// TIA Portal V16 export
// export: Created 2021-11-12T13:31:59.2910616Z, ExportSetting WithDefaults, DisplayName Totally Integrated Automation Portal, DisplayVersion V16 Update 3, DisplayName TIA Portal Version Control Interface, DisplayVersion V16 Update 2, DisplayName TIA Portal Openness, DisplayVersion V16 Update 3, DisplayName SINAMICS Startdrive Advanced, DisplayVersion V16 Update 5, DisplayName SINAMICS Startdrive G130, G150, S120, S150, SINAMICS MV, S210, DisplayVersion V16 Update 5, DisplayName SINAMICS Startdrive G110M, G120, G120C, G120D, G120P, G115D, DisplayVersion V16 Update 5, DisplayName STEP 7 Professional, DisplayVersion V16 Update 3, DisplayName STEP 7 Safety, DisplayVersion V16, DisplayName WinCC UA Professional, DisplayVersion V16 Update 3
FUNCTION_BLOCK "Zone100"   // FB71, LAD
{ S7_Optimized_Access := 'TRUE' }
VERSION : 0.1
// stored: AutoNumber false, IsIECCheckEnabled false, IsRetainMemResEnabled false, MemoryReserve 100, SetENOAutomatically false, UDAEnableTagReadback false
   VAR
      SF_ZoneMode { S7_SetPoint := 'True'} : "STD_Zone";
      SF_StationKAS1Mode { S7_SetPoint := 'True'} : "STD_Station";
      SF_StationKAS2Mode { S7_SetPoint := 'True'} : "STD_Station";
      SF_Station110Mode { S7_SetPoint := 'True'} : "STD_Station";
      SF_Station120Mode { S7_SetPoint := 'True'} : "STD_Station";
      SF_Station1R1Mode { S7_SetPoint := 'True'} : "STD_Station";
      SF_Station1R2Mode { S7_SetPoint := 'True'} : "STD_Station";
      SF_Station130Mode { S7_SetPoint := 'True'} : "STD_Station";
      SF_Station140Mode { S7_SetPoint := 'True'} : "STD_Station";
      SF_Station1R3Mode { S7_SetPoint := 'True'} : "STD_Station";
      SF_Station1R4Mode { S7_SetPoint := 'True'} : "STD_Station";
      SF_Station150Mode { S7_SetPoint := 'True'} : "STD_Station";
      SF_Station160Mode { S7_SetPoint := 'True'} : "STD_Station";
      SF_Station170Mode { S7_SetPoint := 'True'} : "STD_Station";
      SF_Station180Mode { S7_SetPoint := 'True'} : "STD_Station";
      SF_Station1R5Mode { S7_SetPoint := 'True'} : "STD_Station";
      SF_Station1R6Mode { S7_SetPoint := 'True'} : "STD_Station";
      SF_StationBSN1Mode { S7_SetPoint := 'True'} : "STD_Station";
      SF_StationBSN2Mode { S7_SetPoint := 'True'} : "STD_Station";
      SF_CameraLights { S7_SetPoint := 'True'} : "STD_OnOff";
      ST_TONZone1ServModeAct { S7_SetPoint := 'True'} : TON_TIME;   // Timer for Zone 100 service mode
      SS_Edge { S7_SetPoint := 'True'} : Array[0..100] of Bool;
   END_VAR
   VAR_TEMP
      TS_Zone : "UDT_ZoneControl";
      TS_StationKAS1 : "UDT_StationControl";
      TS_StationKAS2 : "UDT_StationControl";
      TS_Station110 : "UDT_StationControl";
      TS_Station120 : "UDT_StationControl";
      TS_Station1R1 : "UDT_StationControl";
      TS_Station1R2 : "UDT_StationControl";
      TS_Station130 : "UDT_StationControl";
      TS_Station140 : "UDT_StationControl";
      TS_Station1R3 : "UDT_StationControl";
      TS_Station1R4 : "UDT_StationControl";
      TS_Station150 : "UDT_StationControl";
      TS_Station160 : "UDT_StationControl";
      TS_Station170 : "UDT_StationControl";
      TS_Station180 : "UDT_StationControl";
      TS_Station1R5 : "UDT_StationControl";
      TS_Station1R6 : "UDT_StationControl";
      TS_StationBSN1 : "UDT_StationControl";
      TS_StationBSN2 : "UDT_StationControl";
      TB1AckFlt1 : Bool;   // LED - acknowledge error button
      TB1AckFlt2 : Bool;   // LED - acknowledge error button
      TB1AckFlt3 : Bool;   // LED - acknowledge error button
      TB1AckSafety1 : Bool;   // LED - acknowledge safety button
      TB1AckSafety2 : Bool;   // LED - acknowledge safety button
      TB1AckSafety3 : Bool;   // LED - acknowledge safety button
      TB1AutStart1 : Bool;   // LED - automat start button
      TB1AutStart2 : Bool;   // LED - automat start button
      TB1AutStart3 : Bool;   // LED - automat start button
      TB1SigRed1 : Bool;   // Light signal - red
      TB1SigRed2 : Bool;   // Light signal - red
      TB1SigRed3 : Bool;   // Light signal - red
      TB1SigYlw1 : Bool;   // Light signal - yellow
      TB1SigYlw2 : Bool;   // Light signal - yellow
      TB1SigYlw3 : Bool;   // Light signal - yellow
      TB1SigGrn1 : Bool;   // Light signal - green
      TB1SigGrn2 : Bool;   // Light signal - green
      TB1SigGrn3 : Bool;   // Light signal - green
      TB1SigAcs1 : Bool;   // Acustic signal
      TB1SigAcs2 : Bool;   // Acustic signal
      TB1SigAcs3 : Bool;   // Acustic signal
      TB1Sig110AutStart : Bool;   // Station 110 run bulb
      TB1Sig110Man : Bool;   // Station 110 manual mode bulb
      TB1Sig110Rem : Bool;   // Station 110 remote mode bulb
      TB1Sig120AutStart : Bool;   // Station 120 run bulb
      TB1Sig120Man : Bool;   // Station 120 manual mode bulb
      TB1Sig120Rem : Bool;   // Station 120 remote mode bulb
      TB1Bin : Bool;   // Something is missing
      TB1CameraLightsON : Bool;
      TB1ReqEndOfCycle : Bool;
      TB1ReqEndOfProd : Bool;
      TB1_1R1AutoOnPE : Bool;   // AutoOn pos edge
      TB1_1R2AutoOnPE : Bool;   // AutoOn pos edge
      TB1_1R3AutoOnPE : Bool;   // AutoOn pos edge
      TB1_1R4AutoOnPE : Bool;   // AutoOn pos edge
      TB1_1R5AutoOnPE : Bool;   // AutoOn pos edge
      TB1_1R6AutoOnPE : Bool;   // AutoOn pos edge
      TB1_1R1AutoOnNE : Bool;   // AutoOn neg edge
      TB1_1R2AutoOnNE : Bool;   // AutoOn neg edge
      TB1_1R3AutoOnNE : Bool;   // AutoOn neg edge
      TB1_1R4AutoOnNE : Bool;   // AutoOn neg edge
      TB1_1R5AutoOnNE : Bool;   // AutoOn neg edge
      TB1_1R6AutoOnNE : Bool;   // AutoOn neg edge
   END_VAR
   VAR_TEMP   // added for the SCL form of the ladder/FBD networks
      _w1 : Bool;
      _w2 : Bool;
      _w3 : Bool;
   END_VAR
BEGIN

REGION Network 1: *************** Zone 100 ***************
END_REGION

REGION Network 2: Zone 100 - Automat switch HMI command from zone to stations
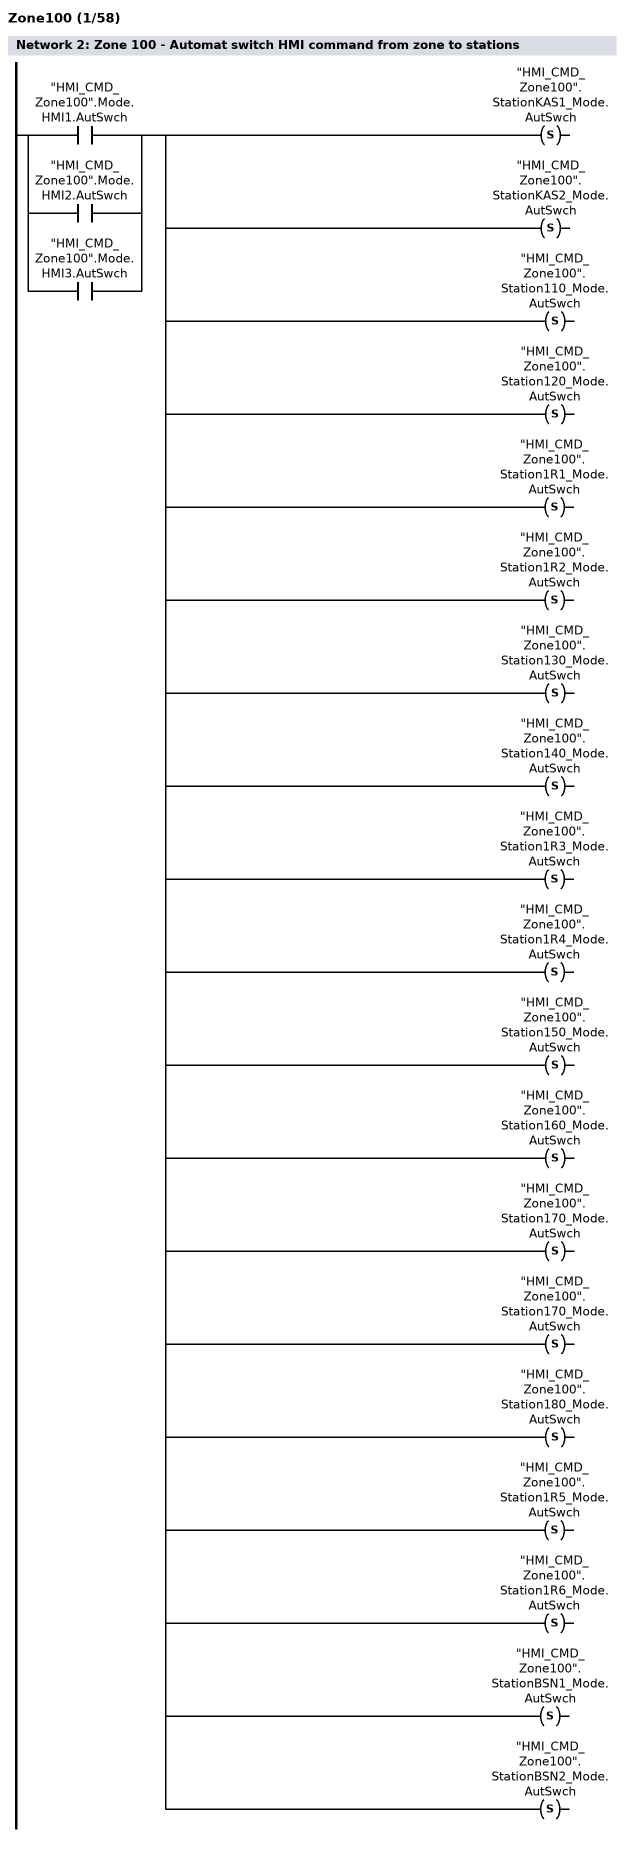
   RUNG wire#powerrail
      Contact( "HMI_CMD_Zone100".Mode.HMI1.AutSwch )
      wire#w1
      S_Coil( "HMI_CMD_Zone100".StationKAS1_Mode.AutSwch )
   END_RUNG
   RUNG wire#powerrail
      Contact( "HMI_CMD_Zone100".Mode.HMI2.AutSwch )
   END_RUNG wire#w1
   RUNG wire#powerrail
      Contact( "HMI_CMD_Zone100".Mode.HMI3.AutSwch )
   END_RUNG wire#w1
   RUNG wire#w1
      S_Coil( "HMI_CMD_Zone100".StationKAS2_Mode.AutSwch )
   END_RUNG
   RUNG wire#w1
      S_Coil( "HMI_CMD_Zone100".Station110_Mode.AutSwch )
   END_RUNG
   RUNG wire#w1
      S_Coil( "HMI_CMD_Zone100".Station120_Mode.AutSwch )
   END_RUNG
   RUNG wire#w1
      S_Coil( "HMI_CMD_Zone100".Station1R1_Mode.AutSwch )
   END_RUNG
   RUNG wire#w1
      S_Coil( "HMI_CMD_Zone100".Station1R2_Mode.AutSwch )
   END_RUNG
   RUNG wire#w1
      S_Coil( "HMI_CMD_Zone100".Station130_Mode.AutSwch )
   END_RUNG
   RUNG wire#w1
      S_Coil( "HMI_CMD_Zone100".Station140_Mode.AutSwch )
   END_RUNG
   RUNG wire#w1
      S_Coil( "HMI_CMD_Zone100".Station1R3_Mode.AutSwch )
   END_RUNG
   RUNG wire#w1
      S_Coil( "HMI_CMD_Zone100".Station1R4_Mode.AutSwch )
   END_RUNG
   RUNG wire#w1
      S_Coil( "HMI_CMD_Zone100".Station150_Mode.AutSwch )
   END_RUNG
   RUNG wire#w1
      S_Coil( "HMI_CMD_Zone100".Station160_Mode.AutSwch )
   END_RUNG
   RUNG wire#w1
      S_Coil( "HMI_CMD_Zone100".Station170_Mode.AutSwch )
   END_RUNG
   RUNG wire#w1
      S_Coil( "HMI_CMD_Zone100".Station170_Mode.AutSwch )
   END_RUNG
   RUNG wire#w1
      S_Coil( "HMI_CMD_Zone100".Station180_Mode.AutSwch )
   END_RUNG
   RUNG wire#w1
      S_Coil( "HMI_CMD_Zone100".Station1R5_Mode.AutSwch )
   END_RUNG
   RUNG wire#w1
      S_Coil( "HMI_CMD_Zone100".Station1R6_Mode.AutSwch )
   END_RUNG
   RUNG wire#w1
      S_Coil( "HMI_CMD_Zone100".StationBSN1_Mode.AutSwch )
   END_RUNG
   RUNG wire#w1
      S_Coil( "HMI_CMD_Zone100".StationBSN2_Mode.AutSwch )
   END_RUNG
   // the same network as SCL:
   IF "HMI_CMD_Zone100".Mode.HMI1.AutSwch OR "HMI_CMD_Zone100".Mode.HMI2.AutSwch OR "HMI_CMD_Zone100".Mode.HMI3.AutSwch THEN
       "HMI_CMD_Zone100".StationKAS1_Mode.AutSwch := TRUE;
       "HMI_CMD_Zone100".StationKAS2_Mode.AutSwch := TRUE;
       "HMI_CMD_Zone100".Station110_Mode.AutSwch := TRUE;
       "HMI_CMD_Zone100".Station120_Mode.AutSwch := TRUE;
       "HMI_CMD_Zone100".Station1R1_Mode.AutSwch := TRUE;
       "HMI_CMD_Zone100".Station1R2_Mode.AutSwch := TRUE;
       "HMI_CMD_Zone100".Station130_Mode.AutSwch := TRUE;
       "HMI_CMD_Zone100".Station140_Mode.AutSwch := TRUE;
       "HMI_CMD_Zone100".Station1R3_Mode.AutSwch := TRUE;
       "HMI_CMD_Zone100".Station1R4_Mode.AutSwch := TRUE;
       "HMI_CMD_Zone100".Station150_Mode.AutSwch := TRUE;
       "HMI_CMD_Zone100".Station160_Mode.AutSwch := TRUE;
       "HMI_CMD_Zone100".Station170_Mode.AutSwch := TRUE;
       "HMI_CMD_Zone100".Station170_Mode.AutSwch := TRUE;
       "HMI_CMD_Zone100".Station180_Mode.AutSwch := TRUE;
       "HMI_CMD_Zone100".Station1R5_Mode.AutSwch := TRUE;
       "HMI_CMD_Zone100".Station1R6_Mode.AutSwch := TRUE;
       "HMI_CMD_Zone100".StationBSN1_Mode.AutSwch := TRUE;
       "HMI_CMD_Zone100".StationBSN2_Mode.AutSwch := TRUE;
   END_IF;
END_REGION

REGION Network 3: Zone 100 - Manual switch HMI command from zone to stations
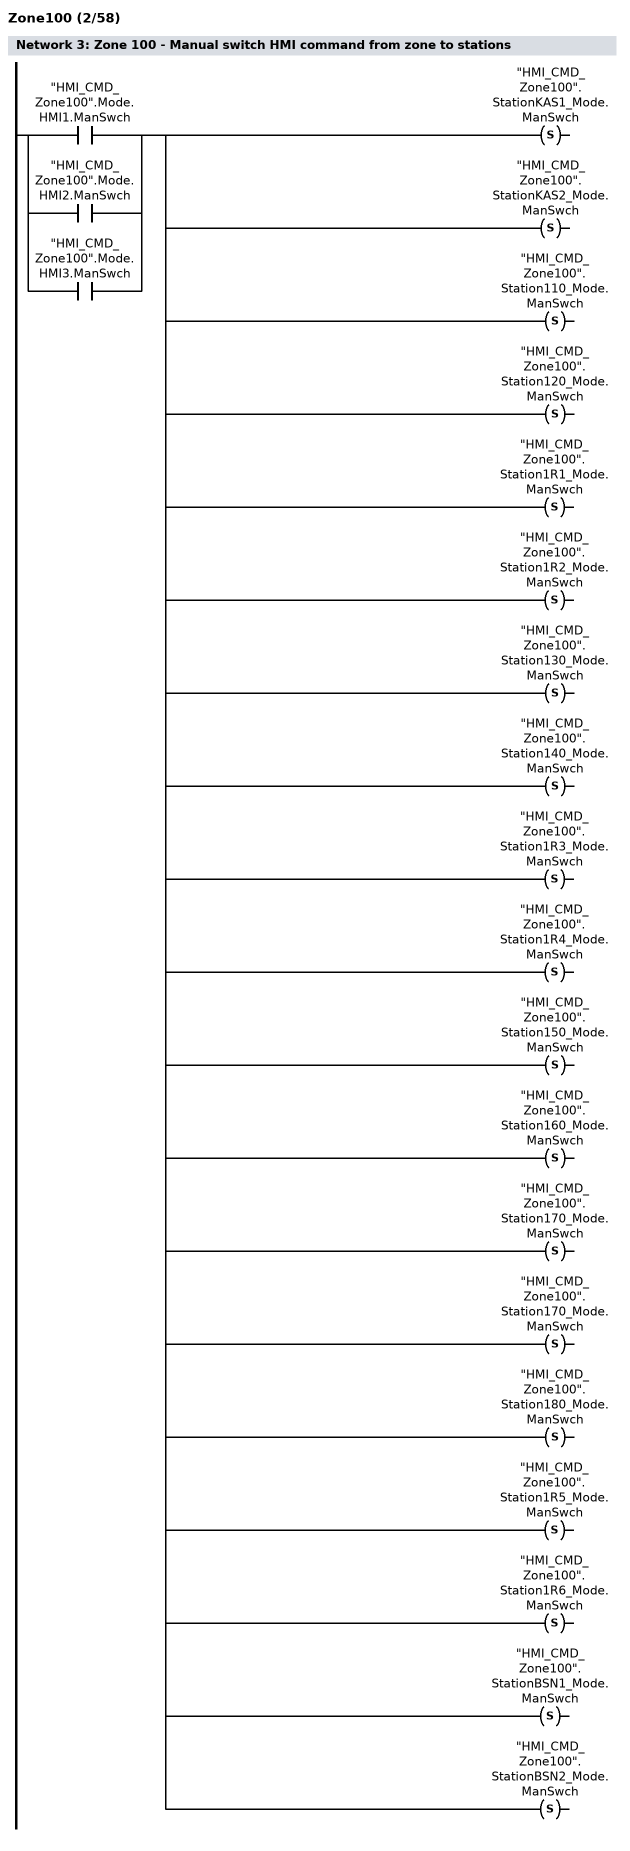
   RUNG wire#powerrail
      Contact( "HMI_CMD_Zone100".Mode.HMI1.ManSwch )
      wire#w1
      S_Coil( "HMI_CMD_Zone100".StationKAS1_Mode.ManSwch )
   END_RUNG
   RUNG wire#powerrail
      Contact( "HMI_CMD_Zone100".Mode.HMI2.ManSwch )
   END_RUNG wire#w1
   RUNG wire#powerrail
      Contact( "HMI_CMD_Zone100".Mode.HMI3.ManSwch )
   END_RUNG wire#w1
   RUNG wire#w1
      S_Coil( "HMI_CMD_Zone100".StationKAS2_Mode.ManSwch )
   END_RUNG
   RUNG wire#w1
      S_Coil( "HMI_CMD_Zone100".Station110_Mode.ManSwch )
   END_RUNG
   RUNG wire#w1
      S_Coil( "HMI_CMD_Zone100".Station120_Mode.ManSwch )
   END_RUNG
   RUNG wire#w1
      S_Coil( "HMI_CMD_Zone100".Station1R1_Mode.ManSwch )
   END_RUNG
   RUNG wire#w1
      S_Coil( "HMI_CMD_Zone100".Station1R2_Mode.ManSwch )
   END_RUNG
   RUNG wire#w1
      S_Coil( "HMI_CMD_Zone100".Station130_Mode.ManSwch )
   END_RUNG
   RUNG wire#w1
      S_Coil( "HMI_CMD_Zone100".Station140_Mode.ManSwch )
   END_RUNG
   RUNG wire#w1
      S_Coil( "HMI_CMD_Zone100".Station1R3_Mode.ManSwch )
   END_RUNG
   RUNG wire#w1
      S_Coil( "HMI_CMD_Zone100".Station1R4_Mode.ManSwch )
   END_RUNG
   RUNG wire#w1
      S_Coil( "HMI_CMD_Zone100".Station150_Mode.ManSwch )
   END_RUNG
   RUNG wire#w1
      S_Coil( "HMI_CMD_Zone100".Station160_Mode.ManSwch )
   END_RUNG
   RUNG wire#w1
      S_Coil( "HMI_CMD_Zone100".Station170_Mode.ManSwch )
   END_RUNG
   RUNG wire#w1
      S_Coil( "HMI_CMD_Zone100".Station170_Mode.ManSwch )
   END_RUNG
   RUNG wire#w1
      S_Coil( "HMI_CMD_Zone100".Station180_Mode.ManSwch )
   END_RUNG
   RUNG wire#w1
      S_Coil( "HMI_CMD_Zone100".Station1R5_Mode.ManSwch )
   END_RUNG
   RUNG wire#w1
      S_Coil( "HMI_CMD_Zone100".Station1R6_Mode.ManSwch )
   END_RUNG
   RUNG wire#w1
      S_Coil( "HMI_CMD_Zone100".StationBSN1_Mode.ManSwch )
   END_RUNG
   RUNG wire#w1
      S_Coil( "HMI_CMD_Zone100".StationBSN2_Mode.ManSwch )
   END_RUNG
   // the same network as SCL:
   IF "HMI_CMD_Zone100".Mode.HMI1.ManSwch OR "HMI_CMD_Zone100".Mode.HMI2.ManSwch OR "HMI_CMD_Zone100".Mode.HMI3.ManSwch THEN
       "HMI_CMD_Zone100".StationKAS1_Mode.ManSwch := TRUE;
       "HMI_CMD_Zone100".StationKAS2_Mode.ManSwch := TRUE;
       "HMI_CMD_Zone100".Station110_Mode.ManSwch := TRUE;
       "HMI_CMD_Zone100".Station120_Mode.ManSwch := TRUE;
       "HMI_CMD_Zone100".Station1R1_Mode.ManSwch := TRUE;
       "HMI_CMD_Zone100".Station1R2_Mode.ManSwch := TRUE;
       "HMI_CMD_Zone100".Station130_Mode.ManSwch := TRUE;
       "HMI_CMD_Zone100".Station140_Mode.ManSwch := TRUE;
       "HMI_CMD_Zone100".Station1R3_Mode.ManSwch := TRUE;
       "HMI_CMD_Zone100".Station1R4_Mode.ManSwch := TRUE;
       "HMI_CMD_Zone100".Station150_Mode.ManSwch := TRUE;
       "HMI_CMD_Zone100".Station160_Mode.ManSwch := TRUE;
       "HMI_CMD_Zone100".Station170_Mode.ManSwch := TRUE;
       "HMI_CMD_Zone100".Station170_Mode.ManSwch := TRUE;
       "HMI_CMD_Zone100".Station180_Mode.ManSwch := TRUE;
       "HMI_CMD_Zone100".Station1R5_Mode.ManSwch := TRUE;
       "HMI_CMD_Zone100".Station1R6_Mode.ManSwch := TRUE;
       "HMI_CMD_Zone100".StationBSN1_Mode.ManSwch := TRUE;
       "HMI_CMD_Zone100".StationBSN2_Mode.ManSwch := TRUE;
   END_IF;
END_REGION

REGION Network 4: Zone 100 - Off switch HMI command from zone to stations
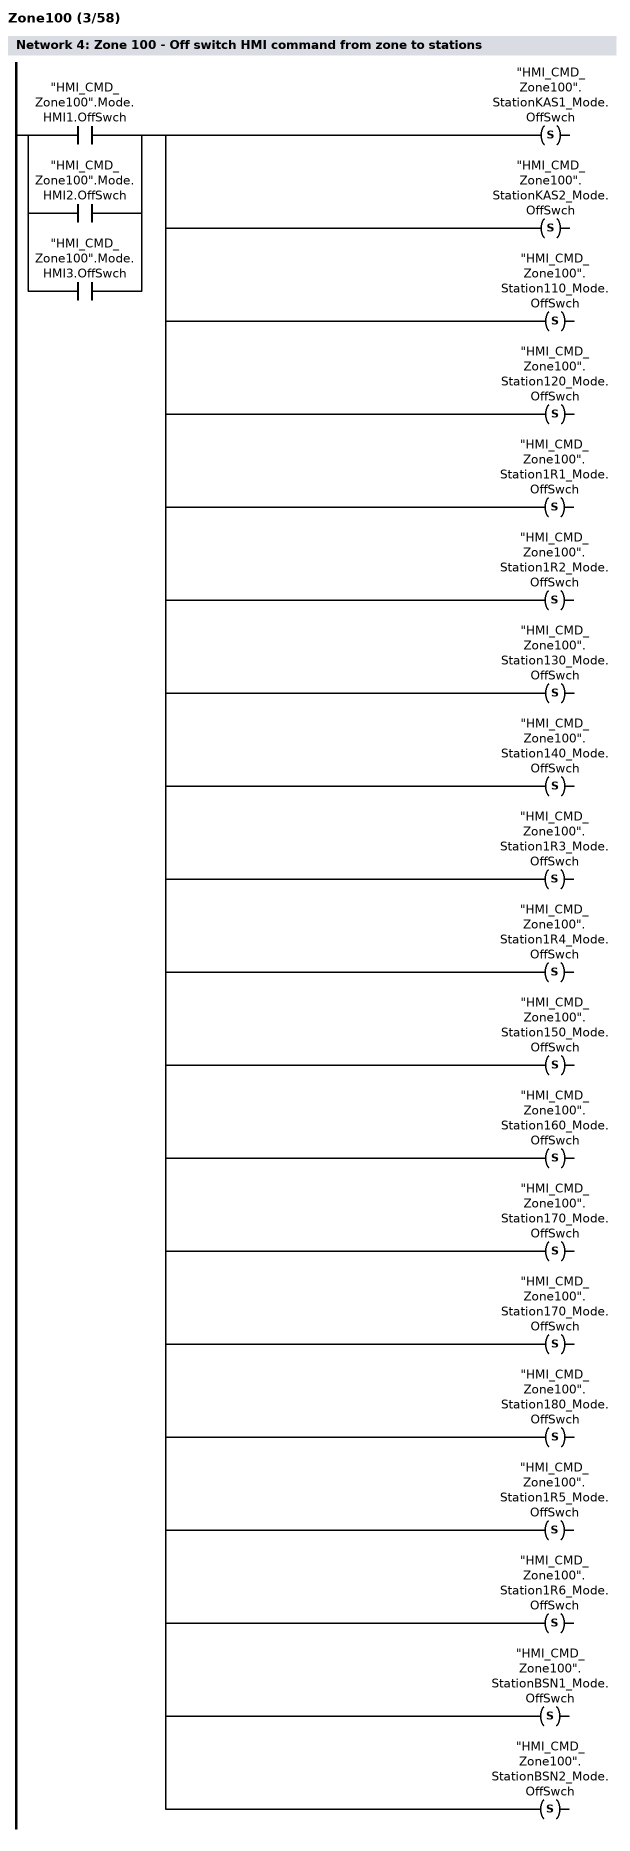
   RUNG wire#powerrail
      Contact( "HMI_CMD_Zone100".Mode.HMI1.OffSwch )
      wire#w1
      S_Coil( "HMI_CMD_Zone100".StationKAS1_Mode.OffSwch )
   END_RUNG
   RUNG wire#powerrail
      Contact( "HMI_CMD_Zone100".Mode.HMI2.OffSwch )
   END_RUNG wire#w1
   RUNG wire#powerrail
      Contact( "HMI_CMD_Zone100".Mode.HMI3.OffSwch )
   END_RUNG wire#w1
   RUNG wire#w1
      S_Coil( "HMI_CMD_Zone100".StationKAS2_Mode.OffSwch )
   END_RUNG
   RUNG wire#w1
      S_Coil( "HMI_CMD_Zone100".Station110_Mode.OffSwch )
   END_RUNG
   RUNG wire#w1
      S_Coil( "HMI_CMD_Zone100".Station120_Mode.OffSwch )
   END_RUNG
   RUNG wire#w1
      S_Coil( "HMI_CMD_Zone100".Station1R1_Mode.OffSwch )
   END_RUNG
   RUNG wire#w1
      S_Coil( "HMI_CMD_Zone100".Station1R2_Mode.OffSwch )
   END_RUNG
   RUNG wire#w1
      S_Coil( "HMI_CMD_Zone100".Station130_Mode.OffSwch )
   END_RUNG
   RUNG wire#w1
      S_Coil( "HMI_CMD_Zone100".Station140_Mode.OffSwch )
   END_RUNG
   RUNG wire#w1
      S_Coil( "HMI_CMD_Zone100".Station1R3_Mode.OffSwch )
   END_RUNG
   RUNG wire#w1
      S_Coil( "HMI_CMD_Zone100".Station1R4_Mode.OffSwch )
   END_RUNG
   RUNG wire#w1
      S_Coil( "HMI_CMD_Zone100".Station150_Mode.OffSwch )
   END_RUNG
   RUNG wire#w1
      S_Coil( "HMI_CMD_Zone100".Station160_Mode.OffSwch )
   END_RUNG
   RUNG wire#w1
      S_Coil( "HMI_CMD_Zone100".Station170_Mode.OffSwch )
   END_RUNG
   RUNG wire#w1
      S_Coil( "HMI_CMD_Zone100".Station170_Mode.OffSwch )
   END_RUNG
   RUNG wire#w1
      S_Coil( "HMI_CMD_Zone100".Station180_Mode.OffSwch )
   END_RUNG
   RUNG wire#w1
      S_Coil( "HMI_CMD_Zone100".Station1R5_Mode.OffSwch )
   END_RUNG
   RUNG wire#w1
      S_Coil( "HMI_CMD_Zone100".Station1R6_Mode.OffSwch )
   END_RUNG
   RUNG wire#w1
      S_Coil( "HMI_CMD_Zone100".StationBSN1_Mode.OffSwch )
   END_RUNG
   RUNG wire#w1
      S_Coil( "HMI_CMD_Zone100".StationBSN2_Mode.OffSwch )
   END_RUNG
   // the same network as SCL:
   IF "HMI_CMD_Zone100".Mode.HMI1.OffSwch OR "HMI_CMD_Zone100".Mode.HMI2.OffSwch OR "HMI_CMD_Zone100".Mode.HMI3.OffSwch THEN
       "HMI_CMD_Zone100".StationKAS1_Mode.OffSwch := TRUE;
       "HMI_CMD_Zone100".StationKAS2_Mode.OffSwch := TRUE;
       "HMI_CMD_Zone100".Station110_Mode.OffSwch := TRUE;
       "HMI_CMD_Zone100".Station120_Mode.OffSwch := TRUE;
       "HMI_CMD_Zone100".Station1R1_Mode.OffSwch := TRUE;
       "HMI_CMD_Zone100".Station1R2_Mode.OffSwch := TRUE;
       "HMI_CMD_Zone100".Station130_Mode.OffSwch := TRUE;
       "HMI_CMD_Zone100".Station140_Mode.OffSwch := TRUE;
       "HMI_CMD_Zone100".Station1R3_Mode.OffSwch := TRUE;
       "HMI_CMD_Zone100".Station1R4_Mode.OffSwch := TRUE;
       "HMI_CMD_Zone100".Station150_Mode.OffSwch := TRUE;
       "HMI_CMD_Zone100".Station160_Mode.OffSwch := TRUE;
       "HMI_CMD_Zone100".Station170_Mode.OffSwch := TRUE;
       "HMI_CMD_Zone100".Station170_Mode.OffSwch := TRUE;
       "HMI_CMD_Zone100".Station180_Mode.OffSwch := TRUE;
       "HMI_CMD_Zone100".Station1R5_Mode.OffSwch := TRUE;
       "HMI_CMD_Zone100".Station1R6_Mode.OffSwch := TRUE;
       "HMI_CMD_Zone100".StationBSN1_Mode.OffSwch := TRUE;
       "HMI_CMD_Zone100".StationBSN2_Mode.OffSwch := TRUE;
   END_IF;
END_REGION

REGION Network 5: Zone 100 - change robot tools command
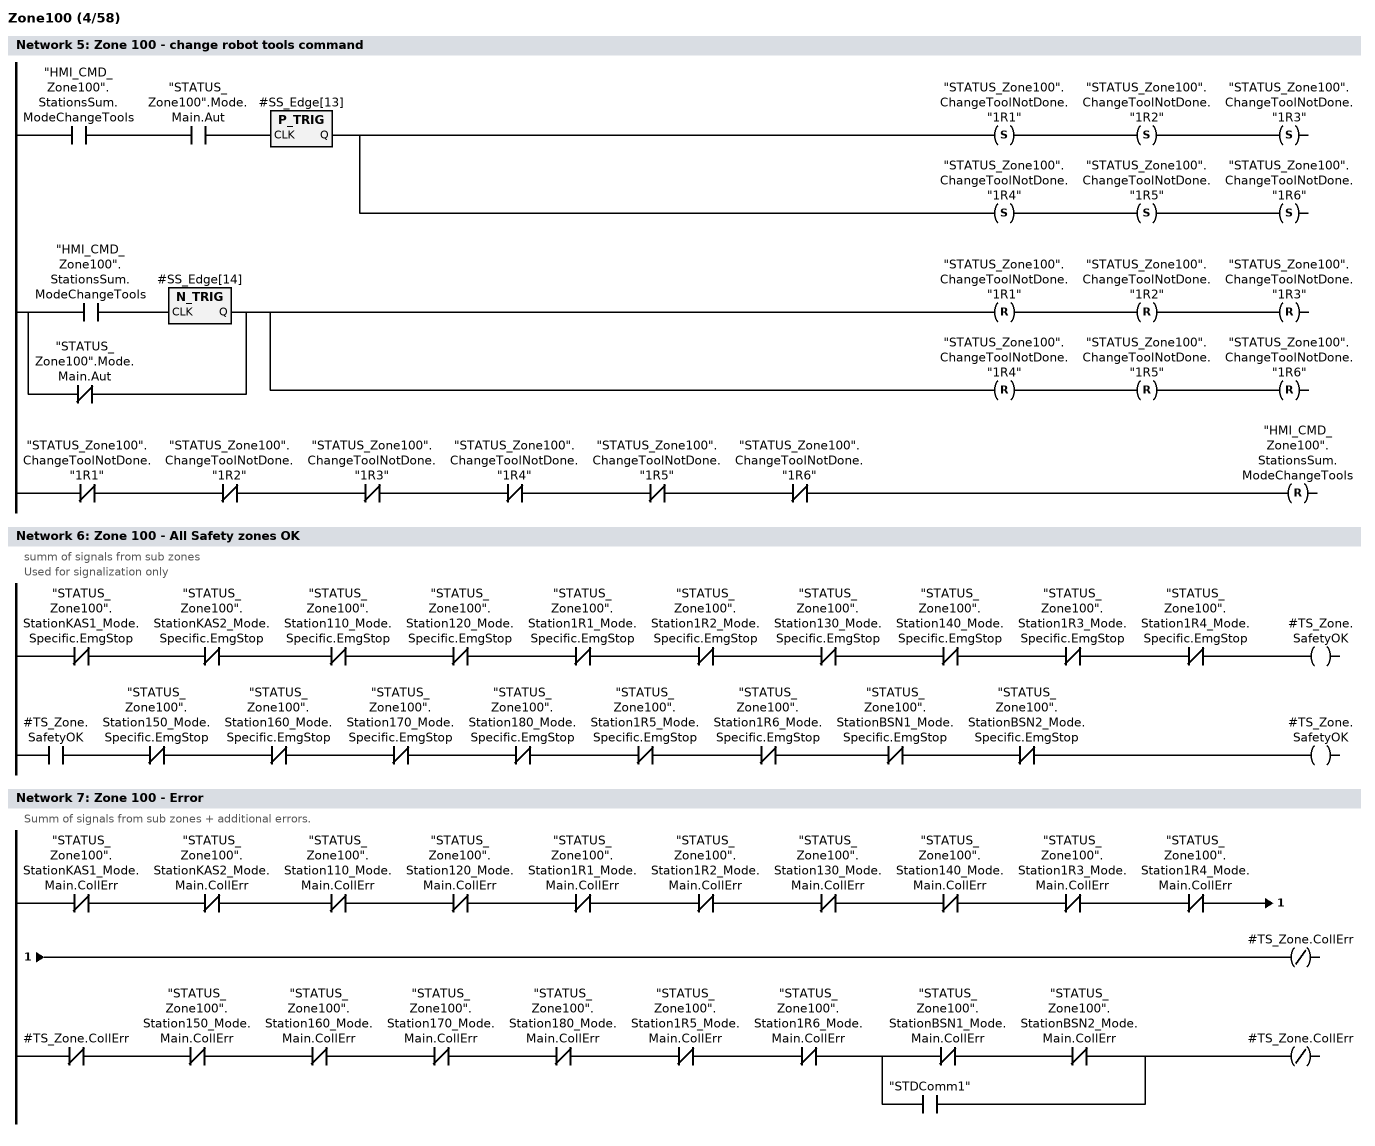
   RUNG wire#powerrail
      Contact( "HMI_CMD_Zone100".StationsSum.ModeChangeTools )
      Contact( "STATUS_Zone100".Mode.Main.Aut )
      P_Trig( #SS_Edge[13] )
      wire#w1
      S_Coil( "STATUS_Zone100".ChangeToolNotDone."1R1" )
      S_Coil( "STATUS_Zone100".ChangeToolNotDone."1R2" )
      S_Coil( "STATUS_Zone100".ChangeToolNotDone."1R3" )
   END_RUNG
   RUNG wire#w1
      S_Coil( "STATUS_Zone100".ChangeToolNotDone."1R4" )
      S_Coil( "STATUS_Zone100".ChangeToolNotDone."1R5" )
      S_Coil( "STATUS_Zone100".ChangeToolNotDone."1R6" )
   END_RUNG
   RUNG wire#powerrail
      Contact( "HMI_CMD_Zone100".StationsSum.ModeChangeTools )
      N_Trig( #SS_Edge[14] )
      wire#w2
      R_Coil( "STATUS_Zone100".ChangeToolNotDone."1R1" )
      R_Coil( "STATUS_Zone100".ChangeToolNotDone."1R2" )
      R_Coil( "STATUS_Zone100".ChangeToolNotDone."1R3" )
   END_RUNG
   RUNG wire#powerrail
      I_Contact( "STATUS_Zone100".Mode.Main.Aut )
   END_RUNG wire#w2
   RUNG wire#w2
      R_Coil( "STATUS_Zone100".ChangeToolNotDone."1R4" )
      R_Coil( "STATUS_Zone100".ChangeToolNotDone."1R5" )
      R_Coil( "STATUS_Zone100".ChangeToolNotDone."1R6" )
   END_RUNG
   RUNG wire#powerrail
      I_Contact( "STATUS_Zone100".ChangeToolNotDone."1R1" )
      I_Contact( "STATUS_Zone100".ChangeToolNotDone."1R2" )
      I_Contact( "STATUS_Zone100".ChangeToolNotDone."1R3" )
      I_Contact( "STATUS_Zone100".ChangeToolNotDone."1R4" )
      I_Contact( "STATUS_Zone100".ChangeToolNotDone."1R5" )
      I_Contact( "STATUS_Zone100".ChangeToolNotDone."1R6" )
      R_Coil( "HMI_CMD_Zone100".StationsSum.ModeChangeTools )
   END_RUNG
   // the same network as SCL:
   #_w1 := "HMI_CMD_Zone100".StationsSum.ModeChangeTools AND "STATUS_Zone100".Mode.Main.Aut;
   #_w2 := #_w1 AND NOT #SS_Edge[13];   // rising edge
   #SS_Edge[13] := #_w1;
   IF #_w2 THEN
       "STATUS_Zone100".ChangeToolNotDone."1R1" := TRUE;
       "STATUS_Zone100".ChangeToolNotDone."1R2" := TRUE;
       "STATUS_Zone100".ChangeToolNotDone."1R3" := TRUE;
       "STATUS_Zone100".ChangeToolNotDone."1R4" := TRUE;
       "STATUS_Zone100".ChangeToolNotDone."1R5" := TRUE;
       "STATUS_Zone100".ChangeToolNotDone."1R6" := TRUE;
   END_IF;
   #_w3 := NOT "HMI_CMD_Zone100".StationsSum.ModeChangeTools AND #SS_Edge[14];   // falling edge
   #SS_Edge[14] := "HMI_CMD_Zone100".StationsSum.ModeChangeTools;
   IF #_w3 OR NOT "STATUS_Zone100".Mode.Main.Aut THEN
       "STATUS_Zone100".ChangeToolNotDone."1R1" := FALSE;
       "STATUS_Zone100".ChangeToolNotDone."1R2" := FALSE;
       "STATUS_Zone100".ChangeToolNotDone."1R3" := FALSE;
       "STATUS_Zone100".ChangeToolNotDone."1R4" := FALSE;
       "STATUS_Zone100".ChangeToolNotDone."1R5" := FALSE;
       "STATUS_Zone100".ChangeToolNotDone."1R6" := FALSE;
   END_IF;
   IF NOT "STATUS_Zone100".ChangeToolNotDone."1R1" AND NOT "STATUS_Zone100".ChangeToolNotDone."1R2" AND NOT "STATUS_Zone100".ChangeToolNotDone."1R3" AND NOT "STATUS_Zone100".ChangeToolNotDone."1R4" AND NOT "STATUS_Zone100".ChangeToolNotDone."1R5" AND NOT "STATUS_Zone100".ChangeToolNotDone."1R6" THEN
       "HMI_CMD_Zone100".StationsSum.ModeChangeTools := FALSE;
   END_IF;
END_REGION

REGION Network 6: Zone 100 - All Safety zones OK
   // summ of signals from sub zones
   // Used for signalization only
   RUNG wire#powerrail
      I_Contact( "STATUS_Zone100".StationKAS1_Mode.Specific.EmgStop )
      I_Contact( "STATUS_Zone100".StationKAS2_Mode.Specific.EmgStop )
      I_Contact( "STATUS_Zone100".Station110_Mode.Specific.EmgStop )
      I_Contact( "STATUS_Zone100".Station120_Mode.Specific.EmgStop )
      I_Contact( "STATUS_Zone100".Station1R1_Mode.Specific.EmgStop )
      I_Contact( "STATUS_Zone100".Station1R2_Mode.Specific.EmgStop )
      I_Contact( "STATUS_Zone100".Station130_Mode.Specific.EmgStop )
      I_Contact( "STATUS_Zone100".Station140_Mode.Specific.EmgStop )
      I_Contact( "STATUS_Zone100".Station1R3_Mode.Specific.EmgStop )
      I_Contact( "STATUS_Zone100".Station1R4_Mode.Specific.EmgStop )
      Coil( #TS_Zone.SafetyOK )
   END_RUNG
   RUNG wire#powerrail
      Contact( #TS_Zone.SafetyOK )
      I_Contact( "STATUS_Zone100".Station150_Mode.Specific.EmgStop )
      I_Contact( "STATUS_Zone100".Station160_Mode.Specific.EmgStop )
      I_Contact( "STATUS_Zone100".Station170_Mode.Specific.EmgStop )
      I_Contact( "STATUS_Zone100".Station180_Mode.Specific.EmgStop )
      I_Contact( "STATUS_Zone100".Station1R5_Mode.Specific.EmgStop )
      I_Contact( "STATUS_Zone100".Station1R6_Mode.Specific.EmgStop )
      I_Contact( "STATUS_Zone100".StationBSN1_Mode.Specific.EmgStop )
      I_Contact( "STATUS_Zone100".StationBSN2_Mode.Specific.EmgStop )
      Coil( #TS_Zone.SafetyOK )
   END_RUNG
   // the same network as SCL:
   #TS_Zone.SafetyOK := NOT "STATUS_Zone100".StationKAS1_Mode.Specific.EmgStop AND NOT "STATUS_Zone100".StationKAS2_Mode.Specific.EmgStop AND NOT "STATUS_Zone100".Station110_Mode.Specific.EmgStop AND NOT "STATUS_Zone100".Station120_Mode.Specific.EmgStop AND NOT "STATUS_Zone100".Station1R1_Mode.Specific.EmgStop AND NOT "STATUS_Zone100".Station1R2_Mode.Specific.EmgStop AND NOT "STATUS_Zone100".Station130_Mode.Specific.EmgStop AND NOT "STATUS_Zone100".Station140_Mode.Specific.EmgStop AND NOT "STATUS_Zone100".Station1R3_Mode.Specific.EmgStop AND NOT "STATUS_Zone100".Station1R4_Mode.Specific.EmgStop;
   #TS_Zone.SafetyOK := #TS_Zone.SafetyOK AND NOT "STATUS_Zone100".Station150_Mode.Specific.EmgStop AND NOT "STATUS_Zone100".Station160_Mode.Specific.EmgStop AND NOT "STATUS_Zone100".Station170_Mode.Specific.EmgStop AND NOT "STATUS_Zone100".Station180_Mode.Specific.EmgStop AND NOT "STATUS_Zone100".Station1R5_Mode.Specific.EmgStop AND NOT "STATUS_Zone100".Station1R6_Mode.Specific.EmgStop AND NOT "STATUS_Zone100".StationBSN1_Mode.Specific.EmgStop AND NOT "STATUS_Zone100".StationBSN2_Mode.Specific.EmgStop;
END_REGION

REGION Network 7: Zone 100 - Error
   // Summ of signals from sub zones + additional errors.
   RUNG wire#powerrail
      I_Contact( "STATUS_Zone100".StationKAS1_Mode.Main.CollErr )
      I_Contact( "STATUS_Zone100".StationKAS2_Mode.Main.CollErr )
      I_Contact( "STATUS_Zone100".Station110_Mode.Main.CollErr )
      I_Contact( "STATUS_Zone100".Station120_Mode.Main.CollErr )
      I_Contact( "STATUS_Zone100".Station1R1_Mode.Main.CollErr )
      I_Contact( "STATUS_Zone100".Station1R2_Mode.Main.CollErr )
      I_Contact( "STATUS_Zone100".Station130_Mode.Main.CollErr )
      I_Contact( "STATUS_Zone100".Station140_Mode.Main.CollErr )
      I_Contact( "STATUS_Zone100".Station1R3_Mode.Main.CollErr )
      I_Contact( "STATUS_Zone100".Station1R4_Mode.Main.CollErr )
      I_Coil( #TS_Zone.CollErr )
   END_RUNG
   RUNG wire#powerrail
      I_Contact( #TS_Zone.CollErr )
      I_Contact( "STATUS_Zone100".Station150_Mode.Main.CollErr )
      I_Contact( "STATUS_Zone100".Station160_Mode.Main.CollErr )
      I_Contact( "STATUS_Zone100".Station170_Mode.Main.CollErr )
      I_Contact( "STATUS_Zone100".Station180_Mode.Main.CollErr )
      I_Contact( "STATUS_Zone100".Station1R5_Mode.Main.CollErr )
      I_Contact( "STATUS_Zone100".Station1R6_Mode.Main.CollErr )
      wire#w1
      I_Contact( "STATUS_Zone100".StationBSN1_Mode.Main.CollErr )
      I_Contact( "STATUS_Zone100".StationBSN2_Mode.Main.CollErr )
      wire#w2
      I_Coil( #TS_Zone.CollErr )
   END_RUNG
   RUNG wire#w1
      Contact( "STDComm1" )
   END_RUNG wire#w2
   // the same network as SCL:
   #TS_Zone.CollErr := NOT (NOT "STATUS_Zone100".StationKAS1_Mode.Main.CollErr AND NOT "STATUS_Zone100".StationKAS2_Mode.Main.CollErr AND NOT "STATUS_Zone100".Station110_Mode.Main.CollErr AND NOT "STATUS_Zone100".Station120_Mode.Main.CollErr AND NOT "STATUS_Zone100".Station1R1_Mode.Main.CollErr AND NOT "STATUS_Zone100".Station1R2_Mode.Main.CollErr AND NOT "STATUS_Zone100".Station130_Mode.Main.CollErr AND NOT "STATUS_Zone100".Station140_Mode.Main.CollErr AND NOT "STATUS_Zone100".Station1R3_Mode.Main.CollErr AND NOT "STATUS_Zone100".Station1R4_Mode.Main.CollErr);
   #TS_Zone.CollErr := NOT (NOT #TS_Zone.CollErr AND NOT "STATUS_Zone100".Station150_Mode.Main.CollErr AND NOT "STATUS_Zone100".Station160_Mode.Main.CollErr AND NOT "STATUS_Zone100".Station170_Mode.Main.CollErr AND NOT "STATUS_Zone100".Station180_Mode.Main.CollErr AND NOT "STATUS_Zone100".Station1R5_Mode.Main.CollErr AND NOT "STATUS_Zone100".Station1R6_Mode.Main.CollErr AND ((NOT "STATUS_Zone100".StationBSN1_Mode.Main.CollErr AND NOT "STATUS_Zone100".StationBSN2_Mode.Main.CollErr) OR "STDComm1"));
END_REGION

REGION Network 8: Zone 100 - Warning
   // Summ of signals from sub zones + additional warnings.
   // Used for signalization only
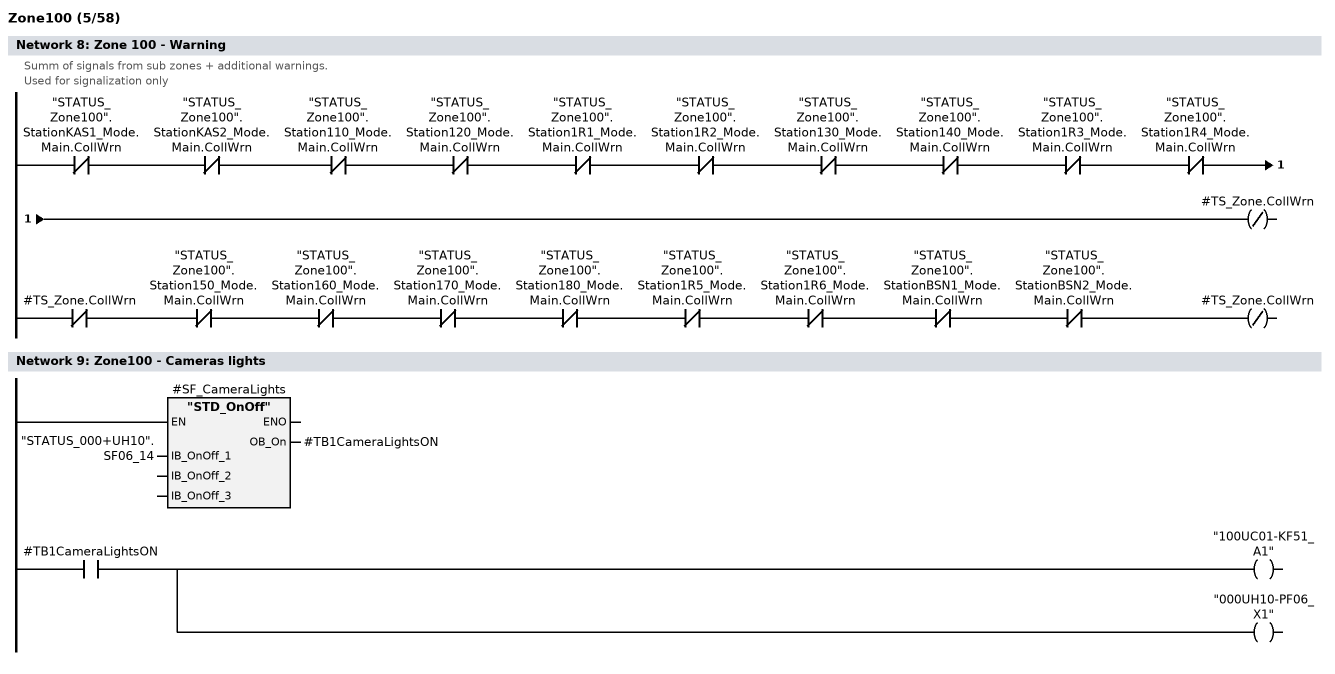
   RUNG wire#powerrail
      I_Contact( "STATUS_Zone100".StationKAS1_Mode.Main.CollWrn )
      I_Contact( "STATUS_Zone100".StationKAS2_Mode.Main.CollWrn )
      I_Contact( "STATUS_Zone100".Station110_Mode.Main.CollWrn )
      I_Contact( "STATUS_Zone100".Station120_Mode.Main.CollWrn )
      I_Contact( "STATUS_Zone100".Station1R1_Mode.Main.CollWrn )
      I_Contact( "STATUS_Zone100".Station1R2_Mode.Main.CollWrn )
      I_Contact( "STATUS_Zone100".Station130_Mode.Main.CollWrn )
      I_Contact( "STATUS_Zone100".Station140_Mode.Main.CollWrn )
      I_Contact( "STATUS_Zone100".Station1R3_Mode.Main.CollWrn )
      I_Contact( "STATUS_Zone100".Station1R4_Mode.Main.CollWrn )
      I_Coil( #TS_Zone.CollWrn )
   END_RUNG
   RUNG wire#powerrail
      I_Contact( #TS_Zone.CollWrn )
      I_Contact( "STATUS_Zone100".Station150_Mode.Main.CollWrn )
      I_Contact( "STATUS_Zone100".Station160_Mode.Main.CollWrn )
      I_Contact( "STATUS_Zone100".Station170_Mode.Main.CollWrn )
      I_Contact( "STATUS_Zone100".Station180_Mode.Main.CollWrn )
      I_Contact( "STATUS_Zone100".Station1R5_Mode.Main.CollWrn )
      I_Contact( "STATUS_Zone100".Station1R6_Mode.Main.CollWrn )
      I_Contact( "STATUS_Zone100".StationBSN1_Mode.Main.CollWrn )
      I_Contact( "STATUS_Zone100".StationBSN2_Mode.Main.CollWrn )
      I_Coil( #TS_Zone.CollWrn )
   END_RUNG
   // the same network as SCL:
   #TS_Zone.CollWrn := NOT (NOT "STATUS_Zone100".StationKAS1_Mode.Main.CollWrn AND NOT "STATUS_Zone100".StationKAS2_Mode.Main.CollWrn AND NOT "STATUS_Zone100".Station110_Mode.Main.CollWrn AND NOT "STATUS_Zone100".Station120_Mode.Main.CollWrn AND NOT "STATUS_Zone100".Station1R1_Mode.Main.CollWrn AND NOT "STATUS_Zone100".Station1R2_Mode.Main.CollWrn AND NOT "STATUS_Zone100".Station130_Mode.Main.CollWrn AND NOT "STATUS_Zone100".Station140_Mode.Main.CollWrn AND NOT "STATUS_Zone100".Station1R3_Mode.Main.CollWrn AND NOT "STATUS_Zone100".Station1R4_Mode.Main.CollWrn);
   #TS_Zone.CollWrn := NOT (NOT #TS_Zone.CollWrn AND NOT "STATUS_Zone100".Station150_Mode.Main.CollWrn AND NOT "STATUS_Zone100".Station160_Mode.Main.CollWrn AND NOT "STATUS_Zone100".Station170_Mode.Main.CollWrn AND NOT "STATUS_Zone100".Station180_Mode.Main.CollWrn AND NOT "STATUS_Zone100".Station1R5_Mode.Main.CollWrn AND NOT "STATUS_Zone100".Station1R6_Mode.Main.CollWrn AND NOT "STATUS_Zone100".StationBSN1_Mode.Main.CollWrn AND NOT "STATUS_Zone100".StationBSN2_Mode.Main.CollWrn);
END_REGION

REGION Network 9: Zone100 - Cameras lights
   RUNG wire#powerrail
      #SF_CameraLights(IB_OnOff_1 := "STATUS_000+UH10".SF06_14, IB_OnOff_2 :=, IB_OnOff_3 :=, OB_On => #TB1CameraLightsON)
   END_RUNG
   RUNG wire#powerrail
      Contact( #TB1CameraLightsON )
      wire#w1
      Coil( "100UC01-KF51_A1" )
   END_RUNG
   RUNG wire#w1
      Coil( "000UH10-PF06_X1" )
   END_RUNG
   // the same network as SCL:
   #SF_CameraLights(IB_OnOff_1 := "STATUS_000+UH10".SF06_14, OB_On => #TB1CameraLightsON);   // "STD_OnOff"
   "100UC01-KF51_A1" := #TB1CameraLightsON;
   "000UH10-PF06_X1" := #TB1CameraLightsON;
END_REGION

REGION Network 10: Zone 100 - All drives running in Automatic
   // Summ of signals from sub zones
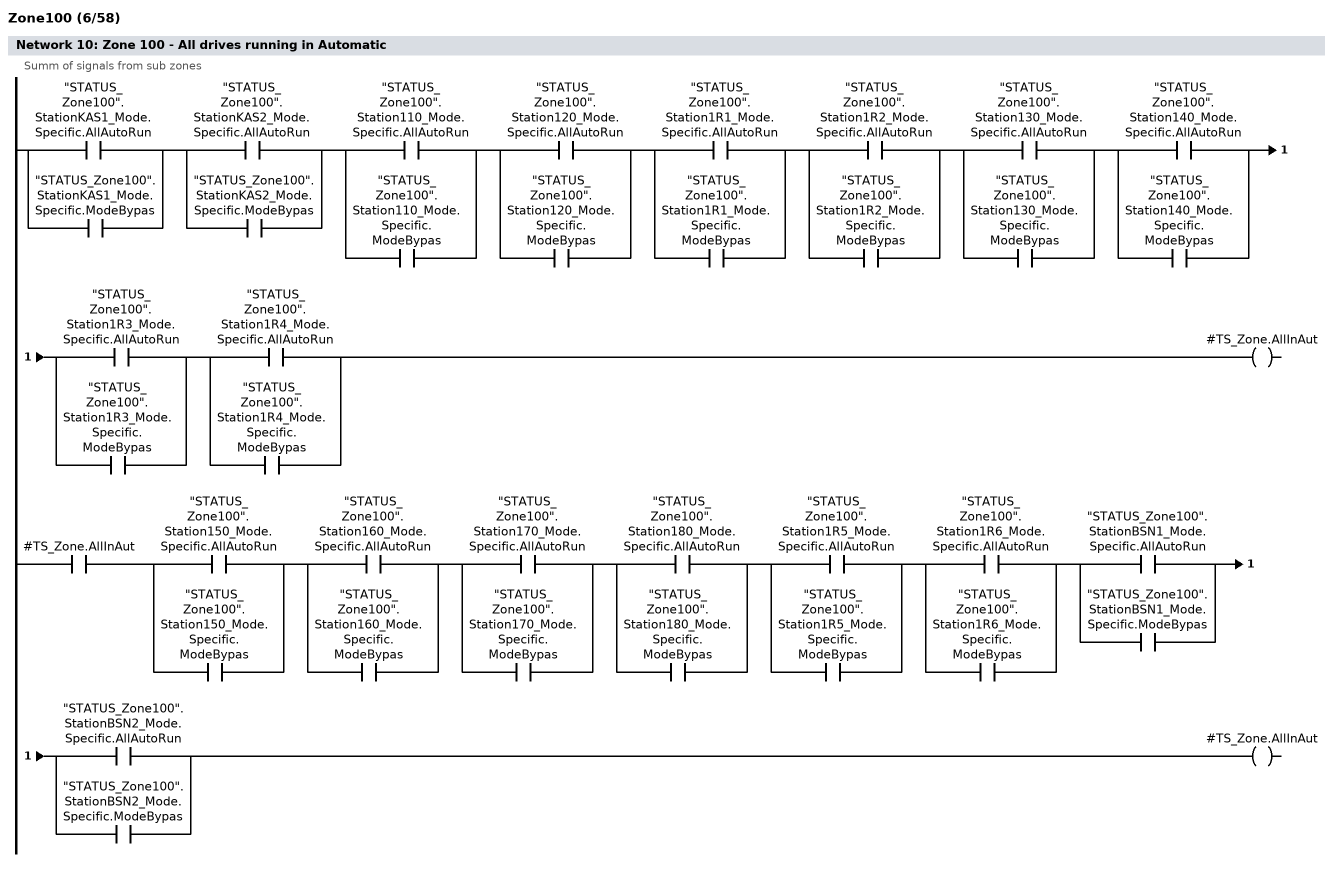
   RUNG wire#powerrail
      Contact( "STATUS_Zone100".StationKAS1_Mode.Specific.AllAutoRun )
      wire#w1
      Contact( "STATUS_Zone100".StationKAS2_Mode.Specific.AllAutoRun )
      wire#w2
      Contact( "STATUS_Zone100".Station110_Mode.Specific.AllAutoRun )
      wire#w3
      Contact( "STATUS_Zone100".Station120_Mode.Specific.AllAutoRun )
      wire#w4
      Contact( "STATUS_Zone100".Station1R1_Mode.Specific.AllAutoRun )
      wire#w5
      Contact( "STATUS_Zone100".Station1R2_Mode.Specific.AllAutoRun )
      wire#w6
      Contact( "STATUS_Zone100".Station130_Mode.Specific.AllAutoRun )
      wire#w7
      Contact( "STATUS_Zone100".Station140_Mode.Specific.AllAutoRun )
      wire#w8
      Contact( "STATUS_Zone100".Station1R3_Mode.Specific.AllAutoRun )
      wire#w9
      Contact( "STATUS_Zone100".Station1R4_Mode.Specific.AllAutoRun )
      wire#w10
      Coil( #TS_Zone.AllInAut )
   END_RUNG
   RUNG wire#powerrail
      Contact( "STATUS_Zone100".StationKAS1_Mode.Specific.ModeBypas )
   END_RUNG wire#w1
   RUNG wire#w1
      Contact( "STATUS_Zone100".StationKAS2_Mode.Specific.ModeBypas )
   END_RUNG wire#w2
   RUNG wire#w2
      Contact( "STATUS_Zone100".Station110_Mode.Specific.ModeBypas )
   END_RUNG wire#w3
   RUNG wire#w3
      Contact( "STATUS_Zone100".Station120_Mode.Specific.ModeBypas )
   END_RUNG wire#w4
   RUNG wire#w4
      Contact( "STATUS_Zone100".Station1R1_Mode.Specific.ModeBypas )
   END_RUNG wire#w5
   RUNG wire#w5
      Contact( "STATUS_Zone100".Station1R2_Mode.Specific.ModeBypas )
   END_RUNG wire#w6
   RUNG wire#w6
      Contact( "STATUS_Zone100".Station130_Mode.Specific.ModeBypas )
   END_RUNG wire#w7
   RUNG wire#w7
      Contact( "STATUS_Zone100".Station140_Mode.Specific.ModeBypas )
   END_RUNG wire#w8
   RUNG wire#w8
      Contact( "STATUS_Zone100".Station1R3_Mode.Specific.ModeBypas )
   END_RUNG wire#w9
   RUNG wire#w9
      Contact( "STATUS_Zone100".Station1R4_Mode.Specific.ModeBypas )
   END_RUNG wire#w10
   RUNG wire#powerrail
      Contact( #TS_Zone.AllInAut )
      wire#w11
      Contact( "STATUS_Zone100".Station150_Mode.Specific.AllAutoRun )
      wire#w12
      Contact( "STATUS_Zone100".Station160_Mode.Specific.AllAutoRun )
      wire#w13
      Contact( "STATUS_Zone100".Station170_Mode.Specific.AllAutoRun )
      wire#w14
      Contact( "STATUS_Zone100".Station180_Mode.Specific.AllAutoRun )
      wire#w15
      Contact( "STATUS_Zone100".Station1R5_Mode.Specific.AllAutoRun )
      wire#w16
      Contact( "STATUS_Zone100".Station1R6_Mode.Specific.AllAutoRun )
      wire#w17
      Contact( "STATUS_Zone100".StationBSN1_Mode.Specific.AllAutoRun )
      wire#w18
      Contact( "STATUS_Zone100".StationBSN2_Mode.Specific.AllAutoRun )
      wire#w19
      Coil( #TS_Zone.AllInAut )
   END_RUNG
   RUNG wire#w11
      Contact( "STATUS_Zone100".Station150_Mode.Specific.ModeBypas )
   END_RUNG wire#w12
   RUNG wire#w12
      Contact( "STATUS_Zone100".Station160_Mode.Specific.ModeBypas )
   END_RUNG wire#w13
   RUNG wire#w13
      Contact( "STATUS_Zone100".Station170_Mode.Specific.ModeBypas )
   END_RUNG wire#w14
   RUNG wire#w14
      Contact( "STATUS_Zone100".Station180_Mode.Specific.ModeBypas )
   END_RUNG wire#w15
   RUNG wire#w15
      Contact( "STATUS_Zone100".Station1R5_Mode.Specific.ModeBypas )
   END_RUNG wire#w16
   RUNG wire#w16
      Contact( "STATUS_Zone100".Station1R6_Mode.Specific.ModeBypas )
   END_RUNG wire#w17
   RUNG wire#w17
      Contact( "STATUS_Zone100".StationBSN1_Mode.Specific.ModeBypas )
   END_RUNG wire#w18
   RUNG wire#w18
      Contact( "STATUS_Zone100".StationBSN2_Mode.Specific.ModeBypas )
   END_RUNG wire#w19
   // the same network as SCL:
   #TS_Zone.AllInAut := ("STATUS_Zone100".StationKAS1_Mode.Specific.AllAutoRun OR "STATUS_Zone100".StationKAS1_Mode.Specific.ModeBypas) AND ("STATUS_Zone100".StationKAS2_Mode.Specific.AllAutoRun OR "STATUS_Zone100".StationKAS2_Mode.Specific.ModeBypas) AND ("STATUS_Zone100".Station110_Mode.Specific.AllAutoRun OR "STATUS_Zone100".Station110_Mode.Specific.ModeBypas) AND ("STATUS_Zone100".Station120_Mode.Specific.AllAutoRun OR "STATUS_Zone100".Station120_Mode.Specific.ModeBypas) AND ("STATUS_Zone100".Station1R1_Mode.Specific.AllAutoRun OR "STATUS_Zone100".Station1R1_Mode.Specific.ModeBypas) AND ("STATUS_Zone100".Station1R2_Mode.Specific.AllAutoRun OR "STATUS_Zone100".Station1R2_Mode.Specific.ModeBypas) AND ("STATUS_Zone100".Station130_Mode.Specific.AllAutoRun OR "STATUS_Zone100".Station130_Mode.Specific.ModeBypas) AND ("STATUS_Zone100".Station140_Mode.Specific.AllAutoRun OR "STATUS_Zone100".Station140_Mode.Specific.ModeBypas) AND ("STATUS_Zone100".Station1R3_Mode.Specific.AllAutoRun OR "STATUS_Zone100".Station1R3_Mode.Specific.ModeBypas) AND ("STATUS_Zone100".Station1R4_Mode.Specific.AllAutoRun OR "STATUS_Zone100".Station1R4_Mode.Specific.ModeBypas);
   #TS_Zone.AllInAut := #TS_Zone.AllInAut AND ("STATUS_Zone100".Station150_Mode.Specific.AllAutoRun OR "STATUS_Zone100".Station150_Mode.Specific.ModeBypas) AND ("STATUS_Zone100".Station160_Mode.Specific.AllAutoRun OR "STATUS_Zone100".Station160_Mode.Specific.ModeBypas) AND ("STATUS_Zone100".Station170_Mode.Specific.AllAutoRun OR "STATUS_Zone100".Station170_Mode.Specific.ModeBypas) AND ("STATUS_Zone100".Station180_Mode.Specific.AllAutoRun OR "STATUS_Zone100".Station180_Mode.Specific.ModeBypas) AND ("STATUS_Zone100".Station1R5_Mode.Specific.AllAutoRun OR "STATUS_Zone100".Station1R5_Mode.Specific.ModeBypas) AND ("STATUS_Zone100".Station1R6_Mode.Specific.AllAutoRun OR "STATUS_Zone100".Station1R6_Mode.Specific.ModeBypas) AND ("STATUS_Zone100".StationBSN1_Mode.Specific.AllAutoRun OR "STATUS_Zone100".StationBSN1_Mode.Specific.ModeBypas) AND ("STATUS_Zone100".StationBSN2_Mode.Specific.AllAutoRun OR "STATUS_Zone100".StationBSN2_Mode.Specific.ModeBypas);
END_REGION

REGION Network 11: Zone 100 - There is some drive that can be started
   // Summ of signals from sub zones.
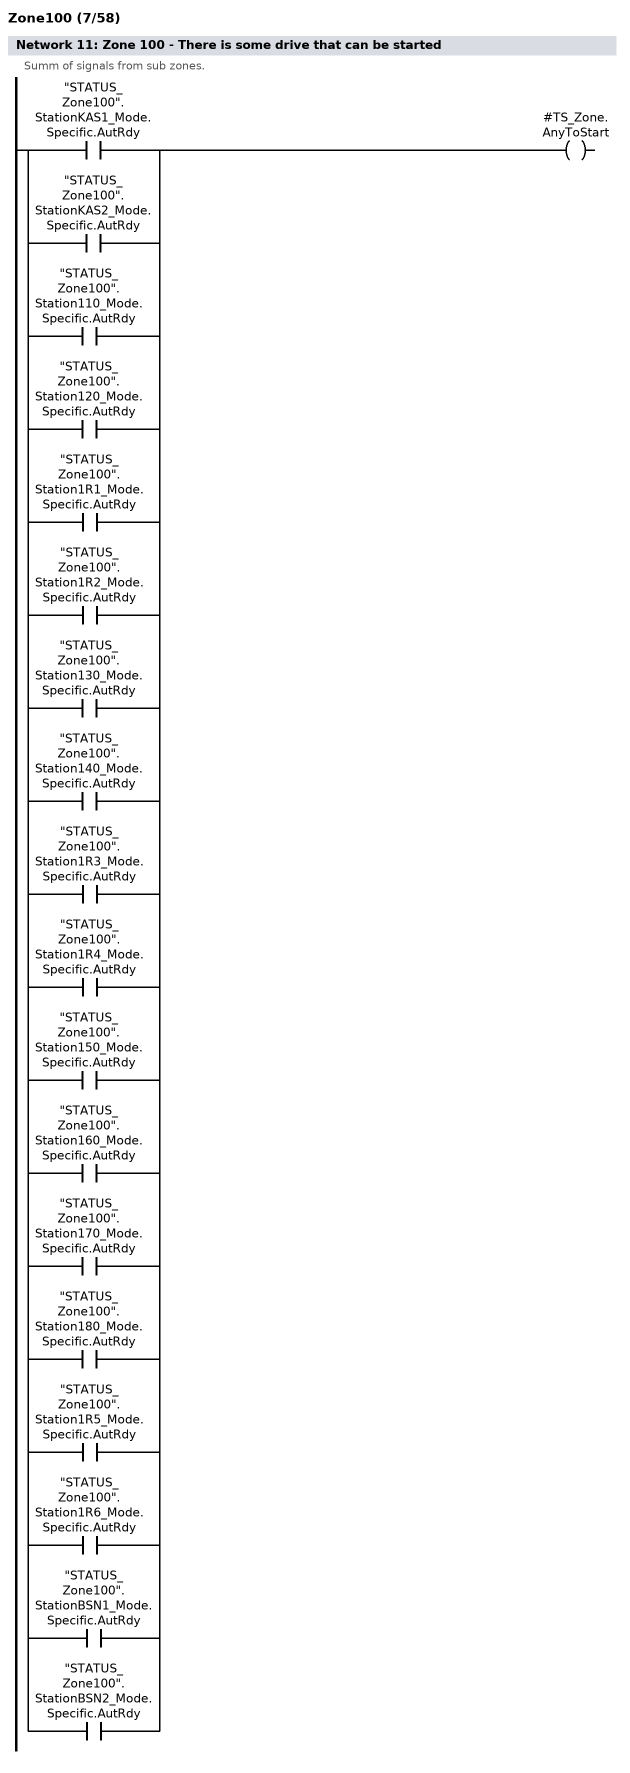
   RUNG wire#powerrail
      Contact( "STATUS_Zone100".StationKAS1_Mode.Specific.AutRdy )
      wire#w1
      Coil( #TS_Zone.AnyToStart )
   END_RUNG
   RUNG wire#powerrail
      Contact( "STATUS_Zone100".StationKAS2_Mode.Specific.AutRdy )
   END_RUNG wire#w1
   RUNG wire#powerrail
      Contact( "STATUS_Zone100".Station110_Mode.Specific.AutRdy )
   END_RUNG wire#w1
   RUNG wire#powerrail
      Contact( "STATUS_Zone100".Station120_Mode.Specific.AutRdy )
   END_RUNG wire#w1
   RUNG wire#powerrail
      Contact( "STATUS_Zone100".Station1R1_Mode.Specific.AutRdy )
   END_RUNG wire#w1
   RUNG wire#powerrail
      Contact( "STATUS_Zone100".Station1R2_Mode.Specific.AutRdy )
   END_RUNG wire#w1
   RUNG wire#powerrail
      Contact( "STATUS_Zone100".Station130_Mode.Specific.AutRdy )
   END_RUNG wire#w1
   RUNG wire#powerrail
      Contact( "STATUS_Zone100".Station140_Mode.Specific.AutRdy )
   END_RUNG wire#w1
   RUNG wire#powerrail
      Contact( "STATUS_Zone100".Station1R3_Mode.Specific.AutRdy )
   END_RUNG wire#w1
   RUNG wire#powerrail
      Contact( "STATUS_Zone100".Station1R4_Mode.Specific.AutRdy )
   END_RUNG wire#w1
   RUNG wire#powerrail
      Contact( "STATUS_Zone100".Station150_Mode.Specific.AutRdy )
   END_RUNG wire#w1
   RUNG wire#powerrail
      Contact( "STATUS_Zone100".Station160_Mode.Specific.AutRdy )
   END_RUNG wire#w1
   RUNG wire#powerrail
      Contact( "STATUS_Zone100".Station170_Mode.Specific.AutRdy )
   END_RUNG wire#w1
   RUNG wire#powerrail
      Contact( "STATUS_Zone100".Station180_Mode.Specific.AutRdy )
   END_RUNG wire#w1
   RUNG wire#powerrail
      Contact( "STATUS_Zone100".Station1R5_Mode.Specific.AutRdy )
   END_RUNG wire#w1
   RUNG wire#powerrail
      Contact( "STATUS_Zone100".Station1R6_Mode.Specific.AutRdy )
   END_RUNG wire#w1
   RUNG wire#powerrail
      Contact( "STATUS_Zone100".StationBSN1_Mode.Specific.AutRdy )
   END_RUNG wire#w1
   RUNG wire#powerrail
      Contact( "STATUS_Zone100".StationBSN2_Mode.Specific.AutRdy )
   END_RUNG wire#w1
   // the same network as SCL:
   #TS_Zone.AnyToStart := "STATUS_Zone100".StationKAS1_Mode.Specific.AutRdy OR "STATUS_Zone100".StationKAS2_Mode.Specific.AutRdy OR "STATUS_Zone100".Station110_Mode.Specific.AutRdy OR "STATUS_Zone100".Station120_Mode.Specific.AutRdy OR "STATUS_Zone100".Station1R1_Mode.Specific.AutRdy OR "STATUS_Zone100".Station1R2_Mode.Specific.AutRdy OR "STATUS_Zone100".Station130_Mode.Specific.AutRdy OR "STATUS_Zone100".Station140_Mode.Specific.AutRdy OR "STATUS_Zone100".Station1R3_Mode.Specific.AutRdy OR "STATUS_Zone100".Station1R4_Mode.Specific.AutRdy OR "STATUS_Zone100".Station150_Mode.Specific.AutRdy OR "STATUS_Zone100".Station160_Mode.Specific.AutRdy OR "STATUS_Zone100".Station170_Mode.Specific.AutRdy OR "STATUS_Zone100".Station180_Mode.Specific.AutRdy OR "STATUS_Zone100".Station1R5_Mode.Specific.AutRdy OR "STATUS_Zone100".Station1R6_Mode.Specific.AutRdy OR "STATUS_Zone100".StationBSN1_Mode.Specific.AutRdy OR "STATUS_Zone100".StationBSN2_Mode.Specific.AutRdy;
END_REGION

REGION Network 12: Zone 100 - Request to suppress alarms from zone
   // This signal is combined with Alarm suppress signal of subzone and
   // sent to electric position
   // When in log 1 new alarms are not generated
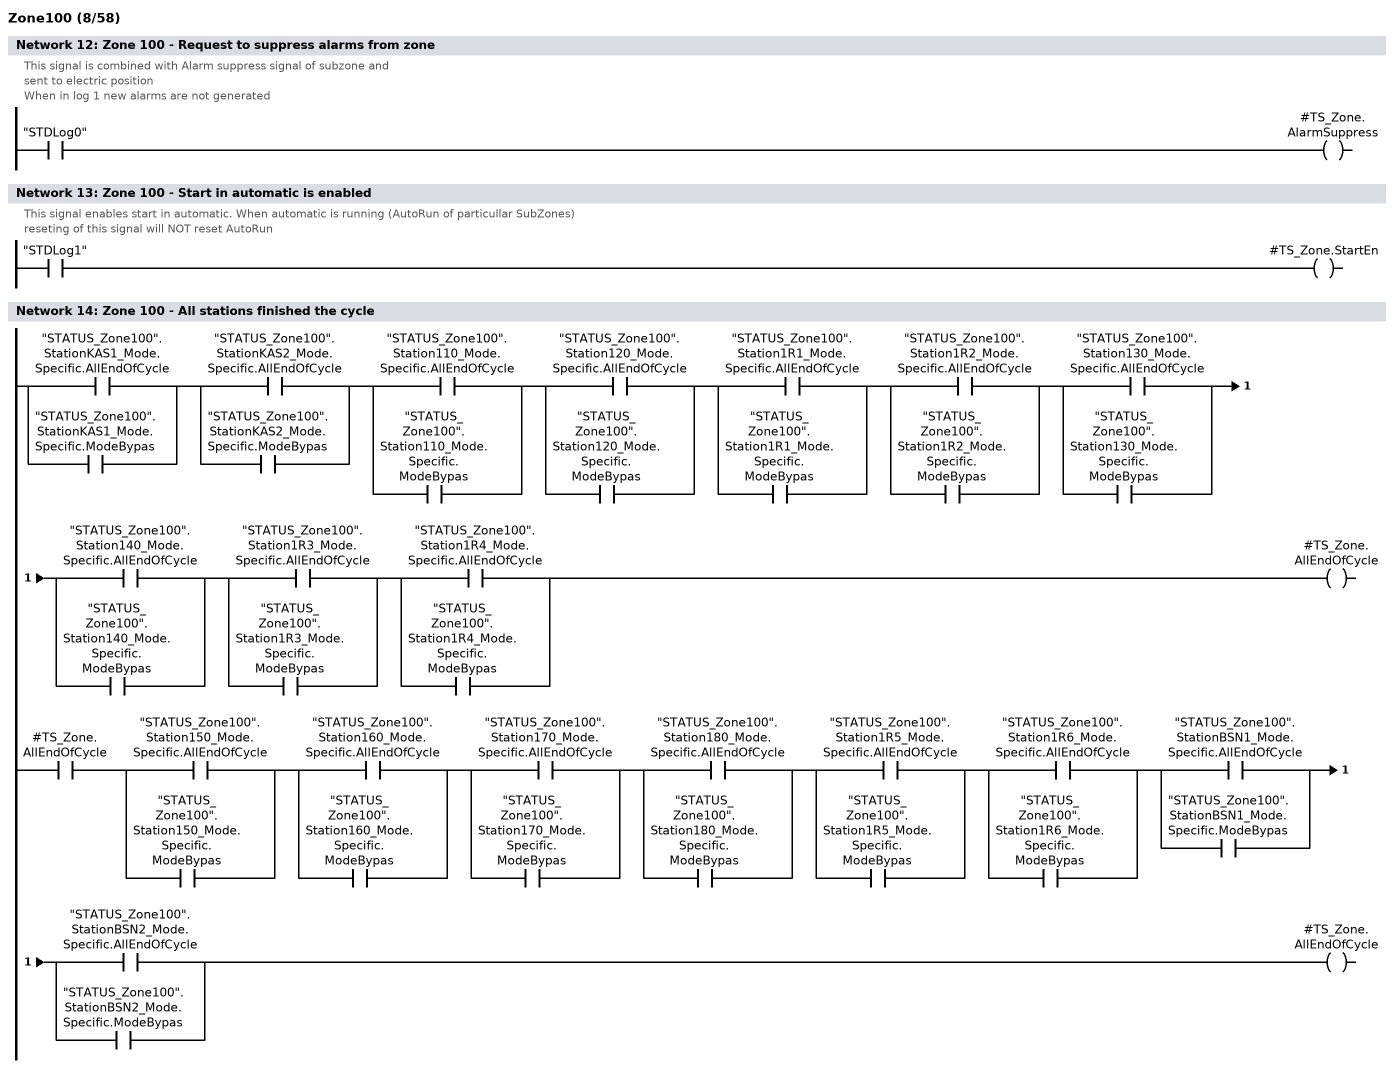
   RUNG wire#powerrail
      Contact( "STDLog0" )
      Coil( #TS_Zone.AlarmSuppress )
   END_RUNG
   // the same network as SCL:
   #TS_Zone.AlarmSuppress := "STDLog0";
END_REGION

REGION Network 13: Zone 100 - Start in automatic is enabled
   // This signal enables start in automatic. When automatic is running (AutoRun of particullar SubZones)
   // reseting of this signal will NOT reset AutoRun
   RUNG wire#powerrail
      Contact( "STDLog1" )
      Coil( #TS_Zone.StartEn )
   END_RUNG
   // the same network as SCL:
   #TS_Zone.StartEn := "STDLog1";
END_REGION

REGION Network 14: Zone 100 - All stations finished the cycle
   RUNG wire#powerrail
      Contact( "STATUS_Zone100".StationKAS1_Mode.Specific.AllEndOfCycle )
      wire#w1
      Contact( "STATUS_Zone100".StationKAS2_Mode.Specific.AllEndOfCycle )
      wire#w2
      Contact( "STATUS_Zone100".Station110_Mode.Specific.AllEndOfCycle )
      wire#w3
      Contact( "STATUS_Zone100".Station120_Mode.Specific.AllEndOfCycle )
      wire#w4
      Contact( "STATUS_Zone100".Station1R1_Mode.Specific.AllEndOfCycle )
      wire#w5
      Contact( "STATUS_Zone100".Station1R2_Mode.Specific.AllEndOfCycle )
      wire#w6
      Contact( "STATUS_Zone100".Station130_Mode.Specific.AllEndOfCycle )
      wire#w7
      Contact( "STATUS_Zone100".Station140_Mode.Specific.AllEndOfCycle )
      wire#w8
      Contact( "STATUS_Zone100".Station1R3_Mode.Specific.AllEndOfCycle )
      wire#w9
      Contact( "STATUS_Zone100".Station1R4_Mode.Specific.AllEndOfCycle )
      wire#w10
      Coil( #TS_Zone.AllEndOfCycle )
   END_RUNG
   RUNG wire#powerrail
      Contact( "STATUS_Zone100".StationKAS1_Mode.Specific.ModeBypas )
   END_RUNG wire#w1
   RUNG wire#w1
      Contact( "STATUS_Zone100".StationKAS2_Mode.Specific.ModeBypas )
   END_RUNG wire#w2
   RUNG wire#w2
      Contact( "STATUS_Zone100".Station110_Mode.Specific.ModeBypas )
   END_RUNG wire#w3
   RUNG wire#w3
      Contact( "STATUS_Zone100".Station120_Mode.Specific.ModeBypas )
   END_RUNG wire#w4
   RUNG wire#w4
      Contact( "STATUS_Zone100".Station1R1_Mode.Specific.ModeBypas )
   END_RUNG wire#w5
   RUNG wire#w5
      Contact( "STATUS_Zone100".Station1R2_Mode.Specific.ModeBypas )
   END_RUNG wire#w6
   RUNG wire#w6
      Contact( "STATUS_Zone100".Station130_Mode.Specific.ModeBypas )
   END_RUNG wire#w7
   RUNG wire#w7
      Contact( "STATUS_Zone100".Station140_Mode.Specific.ModeBypas )
   END_RUNG wire#w8
   RUNG wire#w8
      Contact( "STATUS_Zone100".Station1R3_Mode.Specific.ModeBypas )
   END_RUNG wire#w9
   RUNG wire#w9
      Contact( "STATUS_Zone100".Station1R4_Mode.Specific.ModeBypas )
   END_RUNG wire#w10
   RUNG wire#powerrail
      Contact( #TS_Zone.AllEndOfCycle )
      wire#w11
      Contact( "STATUS_Zone100".Station150_Mode.Specific.AllEndOfCycle )
      wire#w12
      Contact( "STATUS_Zone100".Station160_Mode.Specific.AllEndOfCycle )
      wire#w13
      Contact( "STATUS_Zone100".Station170_Mode.Specific.AllEndOfCycle )
      wire#w14
      Contact( "STATUS_Zone100".Station180_Mode.Specific.AllEndOfCycle )
      wire#w15
      Contact( "STATUS_Zone100".Station1R5_Mode.Specific.AllEndOfCycle )
      wire#w16
      Contact( "STATUS_Zone100".Station1R6_Mode.Specific.AllEndOfCycle )
      wire#w17
      Contact( "STATUS_Zone100".StationBSN1_Mode.Specific.AllEndOfCycle )
      wire#w18
      Contact( "STATUS_Zone100".StationBSN2_Mode.Specific.AllEndOfCycle )
      wire#w19
      Coil( #TS_Zone.AllEndOfCycle )
   END_RUNG
   RUNG wire#w11
      Contact( "STATUS_Zone100".Station150_Mode.Specific.ModeBypas )
   END_RUNG wire#w12
   RUNG wire#w12
      Contact( "STATUS_Zone100".Station160_Mode.Specific.ModeBypas )
   END_RUNG wire#w13
   RUNG wire#w13
      Contact( "STATUS_Zone100".Station170_Mode.Specific.ModeBypas )
   END_RUNG wire#w14
   RUNG wire#w14
      Contact( "STATUS_Zone100".Station180_Mode.Specific.ModeBypas )
   END_RUNG wire#w15
   RUNG wire#w15
      Contact( "STATUS_Zone100".Station1R5_Mode.Specific.ModeBypas )
   END_RUNG wire#w16
   RUNG wire#w16
      Contact( "STATUS_Zone100".Station1R6_Mode.Specific.ModeBypas )
   END_RUNG wire#w17
   RUNG wire#w17
      Contact( "STATUS_Zone100".StationBSN1_Mode.Specific.ModeBypas )
   END_RUNG wire#w18
   RUNG wire#w18
      Contact( "STATUS_Zone100".StationBSN2_Mode.Specific.ModeBypas )
   END_RUNG wire#w19
   // the same network as SCL:
   #TS_Zone.AllEndOfCycle := ("STATUS_Zone100".StationKAS1_Mode.Specific.AllEndOfCycle OR "STATUS_Zone100".StationKAS1_Mode.Specific.ModeBypas) AND ("STATUS_Zone100".StationKAS2_Mode.Specific.AllEndOfCycle OR "STATUS_Zone100".StationKAS2_Mode.Specific.ModeBypas) AND ("STATUS_Zone100".Station110_Mode.Specific.AllEndOfCycle OR "STATUS_Zone100".Station110_Mode.Specific.ModeBypas) AND ("STATUS_Zone100".Station120_Mode.Specific.AllEndOfCycle OR "STATUS_Zone100".Station120_Mode.Specific.ModeBypas) AND ("STATUS_Zone100".Station1R1_Mode.Specific.AllEndOfCycle OR "STATUS_Zone100".Station1R1_Mode.Specific.ModeBypas) AND ("STATUS_Zone100".Station1R2_Mode.Specific.AllEndOfCycle OR "STATUS_Zone100".Station1R2_Mode.Specific.ModeBypas) AND ("STATUS_Zone100".Station130_Mode.Specific.AllEndOfCycle OR "STATUS_Zone100".Station130_Mode.Specific.ModeBypas) AND ("STATUS_Zone100".Station140_Mode.Specific.AllEndOfCycle OR "STATUS_Zone100".Station140_Mode.Specific.ModeBypas) AND ("STATUS_Zone100".Station1R3_Mode.Specific.AllEndOfCycle OR "STATUS_Zone100".Station1R3_Mode.Specific.ModeBypas) AND ("STATUS_Zone100".Station1R4_Mode.Specific.AllEndOfCycle OR "STATUS_Zone100".Station1R4_Mode.Specific.ModeBypas);
   #TS_Zone.AllEndOfCycle := #TS_Zone.AllEndOfCycle AND ("STATUS_Zone100".Station150_Mode.Specific.AllEndOfCycle OR "STATUS_Zone100".Station150_Mode.Specific.ModeBypas) AND ("STATUS_Zone100".Station160_Mode.Specific.AllEndOfCycle OR "STATUS_Zone100".Station160_Mode.Specific.ModeBypas) AND ("STATUS_Zone100".Station170_Mode.Specific.AllEndOfCycle OR "STATUS_Zone100".Station170_Mode.Specific.ModeBypas) AND ("STATUS_Zone100".Station180_Mode.Specific.AllEndOfCycle OR "STATUS_Zone100".Station180_Mode.Specific.ModeBypas) AND ("STATUS_Zone100".Station1R5_Mode.Specific.AllEndOfCycle OR "STATUS_Zone100".Station1R5_Mode.Specific.ModeBypas) AND ("STATUS_Zone100".Station1R6_Mode.Specific.AllEndOfCycle OR "STATUS_Zone100".Station1R6_Mode.Specific.ModeBypas) AND ("STATUS_Zone100".StationBSN1_Mode.Specific.AllEndOfCycle OR "STATUS_Zone100".StationBSN1_Mode.Specific.ModeBypas) AND ("STATUS_Zone100".StationBSN2_Mode.Specific.AllEndOfCycle OR "STATUS_Zone100".StationBSN2_Mode.Specific.ModeBypas);
END_REGION

REGION Network 15: Zone 100 - All stations finished the production
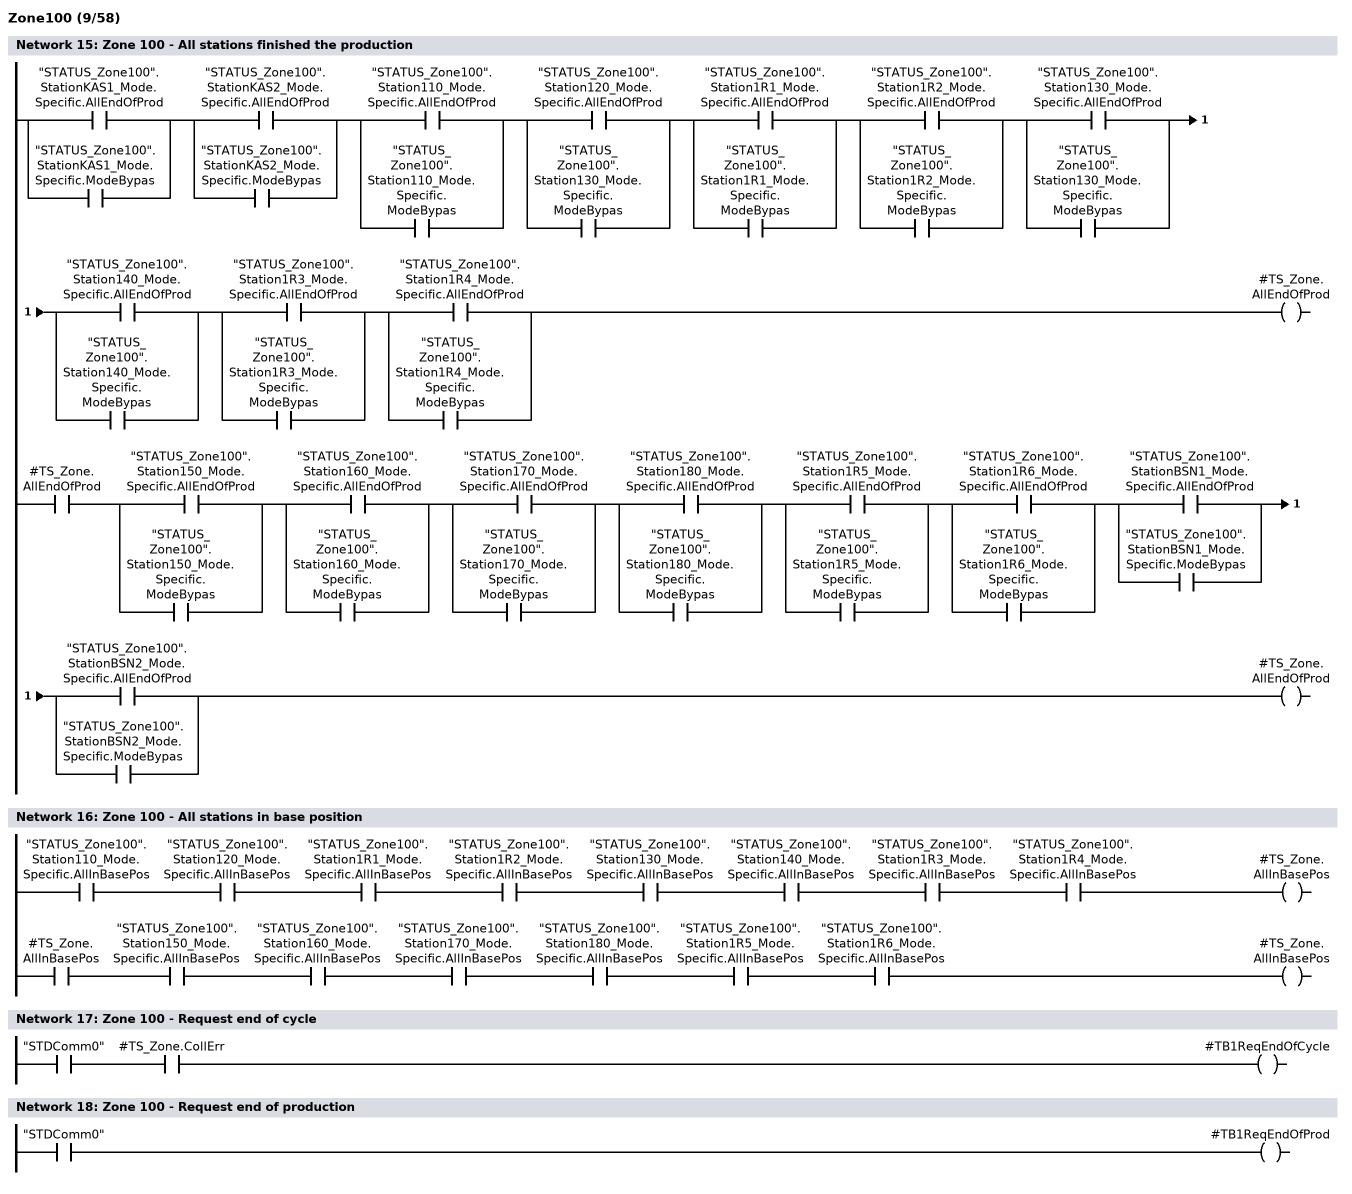
   RUNG wire#powerrail
      Contact( "STATUS_Zone100".StationKAS1_Mode.Specific.AllEndOfProd )
      wire#w1
      Contact( "STATUS_Zone100".StationKAS2_Mode.Specific.AllEndOfProd )
      wire#w2
      Contact( "STATUS_Zone100".Station110_Mode.Specific.AllEndOfProd )
      wire#w3
      Contact( "STATUS_Zone100".Station120_Mode.Specific.AllEndOfProd )
      wire#w4
      Contact( "STATUS_Zone100".Station1R1_Mode.Specific.AllEndOfProd )
      wire#w5
      Contact( "STATUS_Zone100".Station1R2_Mode.Specific.AllEndOfProd )
      wire#w6
      Contact( "STATUS_Zone100".Station130_Mode.Specific.AllEndOfProd )
      wire#w7
      Contact( "STATUS_Zone100".Station140_Mode.Specific.AllEndOfProd )
      wire#w8
      Contact( "STATUS_Zone100".Station1R3_Mode.Specific.AllEndOfProd )
      wire#w9
      Contact( "STATUS_Zone100".Station1R4_Mode.Specific.AllEndOfProd )
      wire#w10
      Coil( #TS_Zone.AllEndOfProd )
   END_RUNG
   RUNG wire#powerrail
      Contact( "STATUS_Zone100".StationKAS1_Mode.Specific.ModeBypas )
   END_RUNG wire#w1
   RUNG wire#w1
      Contact( "STATUS_Zone100".StationKAS2_Mode.Specific.ModeBypas )
   END_RUNG wire#w2
   RUNG wire#w2
      Contact( "STATUS_Zone100".Station110_Mode.Specific.ModeBypas )
   END_RUNG wire#w3
   RUNG wire#w3
      Contact( "STATUS_Zone100".Station130_Mode.Specific.ModeBypas )
   END_RUNG wire#w4
   RUNG wire#w4
      Contact( "STATUS_Zone100".Station1R1_Mode.Specific.ModeBypas )
   END_RUNG wire#w5
   RUNG wire#w5
      Contact( "STATUS_Zone100".Station1R2_Mode.Specific.ModeBypas )
   END_RUNG wire#w6
   RUNG wire#w6
      Contact( "STATUS_Zone100".Station130_Mode.Specific.ModeBypas )
   END_RUNG wire#w7
   RUNG wire#w7
      Contact( "STATUS_Zone100".Station140_Mode.Specific.ModeBypas )
   END_RUNG wire#w8
   RUNG wire#w8
      Contact( "STATUS_Zone100".Station1R3_Mode.Specific.ModeBypas )
   END_RUNG wire#w9
   RUNG wire#w9
      Contact( "STATUS_Zone100".Station1R4_Mode.Specific.ModeBypas )
   END_RUNG wire#w10
   RUNG wire#powerrail
      Contact( #TS_Zone.AllEndOfProd )
      wire#w11
      Contact( "STATUS_Zone100".Station150_Mode.Specific.AllEndOfProd )
      wire#w12
      Contact( "STATUS_Zone100".Station160_Mode.Specific.AllEndOfProd )
      wire#w13
      Contact( "STATUS_Zone100".Station170_Mode.Specific.AllEndOfProd )
      wire#w14
      Contact( "STATUS_Zone100".Station180_Mode.Specific.AllEndOfProd )
      wire#w15
      Contact( "STATUS_Zone100".Station1R5_Mode.Specific.AllEndOfProd )
      wire#w16
      Contact( "STATUS_Zone100".Station1R6_Mode.Specific.AllEndOfProd )
      wire#w17
      Contact( "STATUS_Zone100".StationBSN1_Mode.Specific.AllEndOfProd )
      wire#w18
      Contact( "STATUS_Zone100".StationBSN2_Mode.Specific.AllEndOfProd )
      wire#w19
      Coil( #TS_Zone.AllEndOfProd )
   END_RUNG
   RUNG wire#w11
      Contact( "STATUS_Zone100".Station150_Mode.Specific.ModeBypas )
   END_RUNG wire#w12
   RUNG wire#w12
      Contact( "STATUS_Zone100".Station160_Mode.Specific.ModeBypas )
   END_RUNG wire#w13
   RUNG wire#w13
      Contact( "STATUS_Zone100".Station170_Mode.Specific.ModeBypas )
   END_RUNG wire#w14
   RUNG wire#w14
      Contact( "STATUS_Zone100".Station180_Mode.Specific.ModeBypas )
   END_RUNG wire#w15
   RUNG wire#w15
      Contact( "STATUS_Zone100".Station1R5_Mode.Specific.ModeBypas )
   END_RUNG wire#w16
   RUNG wire#w16
      Contact( "STATUS_Zone100".Station1R6_Mode.Specific.ModeBypas )
   END_RUNG wire#w17
   RUNG wire#w17
      Contact( "STATUS_Zone100".StationBSN1_Mode.Specific.ModeBypas )
   END_RUNG wire#w18
   RUNG wire#w18
      Contact( "STATUS_Zone100".StationBSN2_Mode.Specific.ModeBypas )
   END_RUNG wire#w19
   // the same network as SCL:
   #TS_Zone.AllEndOfProd := ("STATUS_Zone100".StationKAS1_Mode.Specific.AllEndOfProd OR "STATUS_Zone100".StationKAS1_Mode.Specific.ModeBypas) AND ("STATUS_Zone100".StationKAS2_Mode.Specific.AllEndOfProd OR "STATUS_Zone100".StationKAS2_Mode.Specific.ModeBypas) AND ("STATUS_Zone100".Station110_Mode.Specific.AllEndOfProd OR "STATUS_Zone100".Station110_Mode.Specific.ModeBypas) AND ("STATUS_Zone100".Station120_Mode.Specific.AllEndOfProd OR "STATUS_Zone100".Station130_Mode.Specific.ModeBypas) AND ("STATUS_Zone100".Station1R1_Mode.Specific.AllEndOfProd OR "STATUS_Zone100".Station1R1_Mode.Specific.ModeBypas) AND ("STATUS_Zone100".Station1R2_Mode.Specific.AllEndOfProd OR "STATUS_Zone100".Station1R2_Mode.Specific.ModeBypas) AND ("STATUS_Zone100".Station130_Mode.Specific.AllEndOfProd OR "STATUS_Zone100".Station130_Mode.Specific.ModeBypas) AND ("STATUS_Zone100".Station140_Mode.Specific.AllEndOfProd OR "STATUS_Zone100".Station140_Mode.Specific.ModeBypas) AND ("STATUS_Zone100".Station1R3_Mode.Specific.AllEndOfProd OR "STATUS_Zone100".Station1R3_Mode.Specific.ModeBypas) AND ("STATUS_Zone100".Station1R4_Mode.Specific.AllEndOfProd OR "STATUS_Zone100".Station1R4_Mode.Specific.ModeBypas);
   #TS_Zone.AllEndOfProd := #TS_Zone.AllEndOfProd AND ("STATUS_Zone100".Station150_Mode.Specific.AllEndOfProd OR "STATUS_Zone100".Station150_Mode.Specific.ModeBypas) AND ("STATUS_Zone100".Station160_Mode.Specific.AllEndOfProd OR "STATUS_Zone100".Station160_Mode.Specific.ModeBypas) AND ("STATUS_Zone100".Station170_Mode.Specific.AllEndOfProd OR "STATUS_Zone100".Station170_Mode.Specific.ModeBypas) AND ("STATUS_Zone100".Station180_Mode.Specific.AllEndOfProd OR "STATUS_Zone100".Station180_Mode.Specific.ModeBypas) AND ("STATUS_Zone100".Station1R5_Mode.Specific.AllEndOfProd OR "STATUS_Zone100".Station1R5_Mode.Specific.ModeBypas) AND ("STATUS_Zone100".Station1R6_Mode.Specific.AllEndOfProd OR "STATUS_Zone100".Station1R6_Mode.Specific.ModeBypas) AND ("STATUS_Zone100".StationBSN1_Mode.Specific.AllEndOfProd OR "STATUS_Zone100".StationBSN1_Mode.Specific.ModeBypas) AND ("STATUS_Zone100".StationBSN2_Mode.Specific.AllEndOfProd OR "STATUS_Zone100".StationBSN2_Mode.Specific.ModeBypas);
END_REGION

REGION Network 16: Zone 100 - All stations in base position
   RUNG wire#powerrail
      Contact( "STATUS_Zone100".Station110_Mode.Specific.AllInBasePos )
      Contact( "STATUS_Zone100".Station120_Mode.Specific.AllInBasePos )
      Contact( "STATUS_Zone100".Station1R1_Mode.Specific.AllInBasePos )
      Contact( "STATUS_Zone100".Station1R2_Mode.Specific.AllInBasePos )
      Contact( "STATUS_Zone100".Station130_Mode.Specific.AllInBasePos )
      Contact( "STATUS_Zone100".Station140_Mode.Specific.AllInBasePos )
      Contact( "STATUS_Zone100".Station1R3_Mode.Specific.AllInBasePos )
      Contact( "STATUS_Zone100".Station1R4_Mode.Specific.AllInBasePos )
      Coil( #TS_Zone.AllInBasePos )
   END_RUNG
   RUNG wire#powerrail
      Contact( #TS_Zone.AllInBasePos )
      Contact( "STATUS_Zone100".Station150_Mode.Specific.AllInBasePos )
      Contact( "STATUS_Zone100".Station160_Mode.Specific.AllInBasePos )
      Contact( "STATUS_Zone100".Station170_Mode.Specific.AllInBasePos )
      Contact( "STATUS_Zone100".Station180_Mode.Specific.AllInBasePos )
      Contact( "STATUS_Zone100".Station1R5_Mode.Specific.AllInBasePos )
      Contact( "STATUS_Zone100".Station1R6_Mode.Specific.AllInBasePos )
      Coil( #TS_Zone.AllInBasePos )
   END_RUNG
   // the same network as SCL:
   #TS_Zone.AllInBasePos := "STATUS_Zone100".Station110_Mode.Specific.AllInBasePos AND "STATUS_Zone100".Station120_Mode.Specific.AllInBasePos AND "STATUS_Zone100".Station1R1_Mode.Specific.AllInBasePos AND "STATUS_Zone100".Station1R2_Mode.Specific.AllInBasePos AND "STATUS_Zone100".Station130_Mode.Specific.AllInBasePos AND "STATUS_Zone100".Station140_Mode.Specific.AllInBasePos AND "STATUS_Zone100".Station1R3_Mode.Specific.AllInBasePos AND "STATUS_Zone100".Station1R4_Mode.Specific.AllInBasePos;
   #TS_Zone.AllInBasePos := #TS_Zone.AllInBasePos AND "STATUS_Zone100".Station150_Mode.Specific.AllInBasePos AND "STATUS_Zone100".Station160_Mode.Specific.AllInBasePos AND "STATUS_Zone100".Station170_Mode.Specific.AllInBasePos AND "STATUS_Zone100".Station180_Mode.Specific.AllInBasePos AND "STATUS_Zone100".Station1R5_Mode.Specific.AllInBasePos AND "STATUS_Zone100".Station1R6_Mode.Specific.AllInBasePos;
END_REGION

REGION Network 17: Zone 100 - Request end of cycle
   RUNG wire#powerrail
      Contact( "STDComm0" )
      Contact( #TS_Zone.CollErr )
      Coil( #TB1ReqEndOfCycle )
   END_RUNG
   // the same network as SCL:
   #TB1ReqEndOfCycle := "STDComm0" AND #TS_Zone.CollErr;
END_REGION

REGION Network 18: Zone 100 - Request end of production
   RUNG wire#powerrail
      Contact( "STDComm0" )
      Coil( #TB1ReqEndOfProd )
   END_RUNG
   // the same network as SCL:
   #TB1ReqEndOfProd := "STDComm0";
END_REGION

REGION Network 19: Zone 100 - Number of selected devices
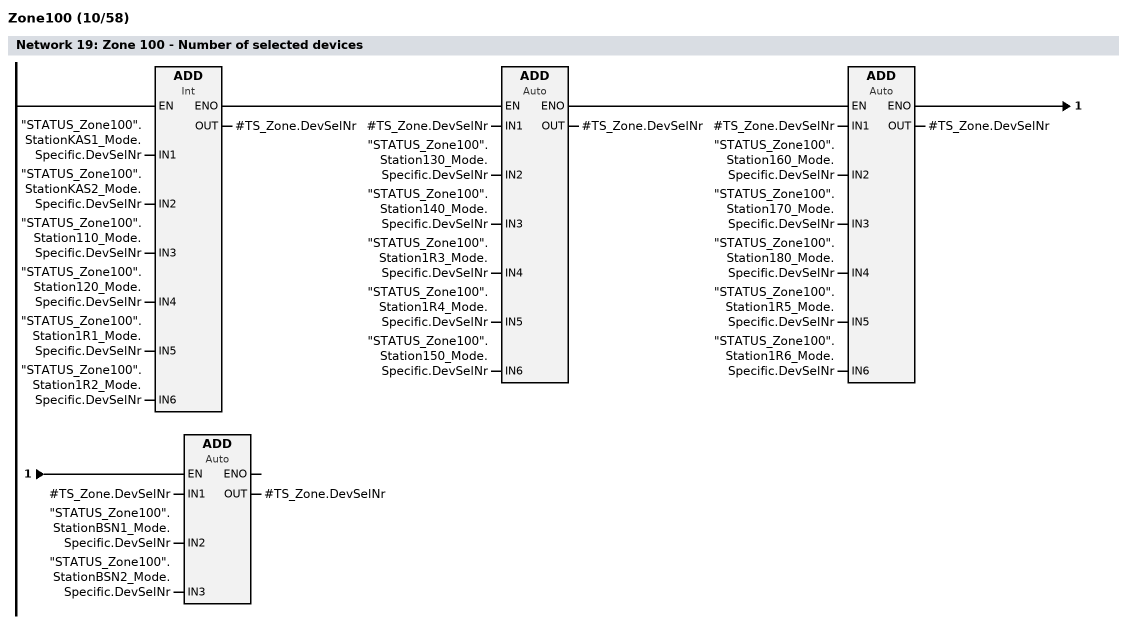
   RUNG wire#powerrail
      { S7_Templates := "SrcType := Int" } Add(in1 := "STATUS_Zone100".StationKAS1_Mode.Specific.DevSelNr, in2 := "STATUS_Zone100".StationKAS2_Mode.Specific.DevSelNr, in3 := "STATUS_Zone100".Station110_Mode.Specific.DevSelNr, in4 := "STATUS_Zone100".Station120_Mode.Specific.DevSelNr, in5 := "STATUS_Zone100".Station1R1_Mode.Specific.DevSelNr, in6 := "STATUS_Zone100".Station1R2_Mode.Specific.DevSelNr, out => #TS_Zone.DevSelNr)
      Add(in1 := #TS_Zone.DevSelNr, in2 := "STATUS_Zone100".Station130_Mode.Specific.DevSelNr, in3 := "STATUS_Zone100".Station140_Mode.Specific.DevSelNr, in4 := "STATUS_Zone100".Station1R3_Mode.Specific.DevSelNr, in5 := "STATUS_Zone100".Station1R4_Mode.Specific.DevSelNr, in6 := "STATUS_Zone100".Station150_Mode.Specific.DevSelNr, out => #TS_Zone.DevSelNr)
      Add(in1 := #TS_Zone.DevSelNr, in2 := "STATUS_Zone100".Station160_Mode.Specific.DevSelNr, in3 := "STATUS_Zone100".Station170_Mode.Specific.DevSelNr, in4 := "STATUS_Zone100".Station180_Mode.Specific.DevSelNr, in5 := "STATUS_Zone100".Station1R5_Mode.Specific.DevSelNr, in6 := "STATUS_Zone100".Station1R6_Mode.Specific.DevSelNr, out => #TS_Zone.DevSelNr)
      Add(in1 := #TS_Zone.DevSelNr, in2 := "STATUS_Zone100".StationBSN1_Mode.Specific.DevSelNr, in3 := "STATUS_Zone100".StationBSN2_Mode.Specific.DevSelNr, out => #TS_Zone.DevSelNr)
   END_RUNG
   // the same network as SCL:
   #TS_Zone.DevSelNr := "STATUS_Zone100".StationKAS1_Mode.Specific.DevSelNr + "STATUS_Zone100".StationKAS2_Mode.Specific.DevSelNr + "STATUS_Zone100".Station110_Mode.Specific.DevSelNr + "STATUS_Zone100".Station120_Mode.Specific.DevSelNr + "STATUS_Zone100".Station1R1_Mode.Specific.DevSelNr + "STATUS_Zone100".Station1R2_Mode.Specific.DevSelNr;
   #TS_Zone.DevSelNr := #TS_Zone.DevSelNr + "STATUS_Zone100".Station130_Mode.Specific.DevSelNr + "STATUS_Zone100".Station140_Mode.Specific.DevSelNr + "STATUS_Zone100".Station1R3_Mode.Specific.DevSelNr + "STATUS_Zone100".Station1R4_Mode.Specific.DevSelNr + "STATUS_Zone100".Station150_Mode.Specific.DevSelNr;
   #TS_Zone.DevSelNr := #TS_Zone.DevSelNr + "STATUS_Zone100".Station160_Mode.Specific.DevSelNr + "STATUS_Zone100".Station170_Mode.Specific.DevSelNr + "STATUS_Zone100".Station180_Mode.Specific.DevSelNr + "STATUS_Zone100".Station1R5_Mode.Specific.DevSelNr + "STATUS_Zone100".Station1R6_Mode.Specific.DevSelNr;
   #TS_Zone.DevSelNr := #TS_Zone.DevSelNr + "STATUS_Zone100".StationBSN1_Mode.Specific.DevSelNr + "STATUS_Zone100".StationBSN2_Mode.Specific.DevSelNr;
END_REGION

REGION Network 20: Zone 100 - Main control
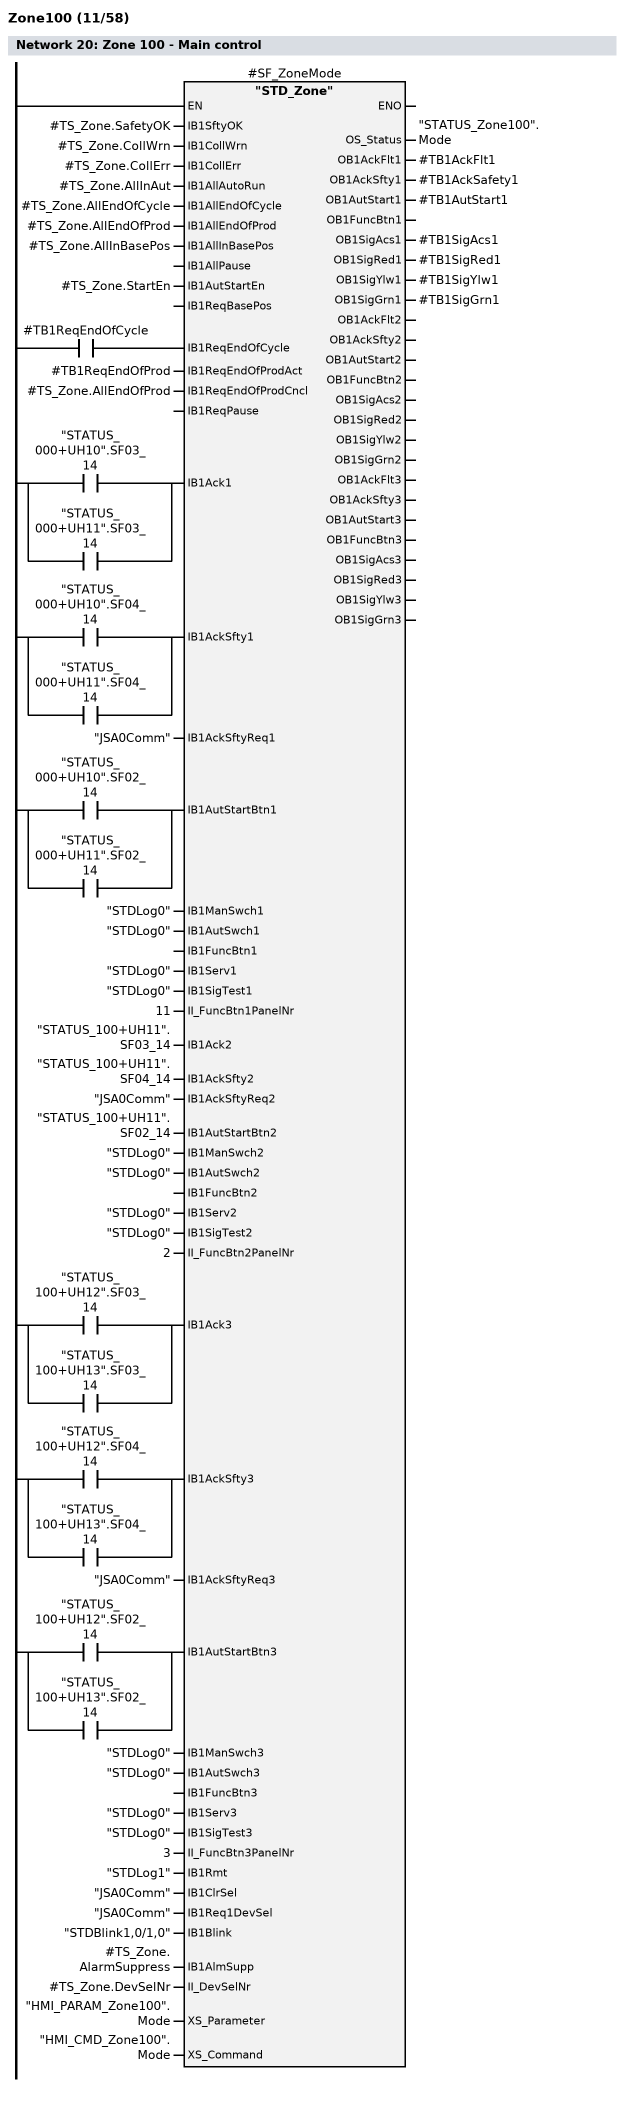
   RUNG wire#powerrail
      #SF_ZoneMode(IB1ReqEndOfCycle := wire#w1, IB1Ack1 := wire#w2, IB1AckSfty1 := wire#w3, IB1AutStartBtn1 := wire#w4, IB1Ack3 := wire#w5, IB1AckSfty3 := wire#w6, IB1AutStartBtn3 := wire#w7, IB1SftyOK := #TS_Zone.SafetyOK, IB1CollWrn := #TS_Zone.CollWrn, IB1CollErr := #TS_Zone.CollErr, IB1AllAutoRun := #TS_Zone.AllInAut, IB1AllEndOfCycle := #TS_Zone.AllEndOfCycle, IB1AllEndOfProd := #TS_Zone.AllEndOfProd, IB1AllInBasePos := #TS_Zone.AllInBasePos, IB1AllPause :=, IB1AutStartEn := #TS_Zone.StartEn, IB1ReqBasePos :=, IB1ReqEndOfProdAct := #TB1ReqEndOfProd, IB1ReqEndOfProdCncl := #TS_Zone.AllEndOfProd, IB1ReqPause :=, IB1AckSftyReq1 := "JSA0Comm", IB1ManSwch1 := "STDLog0", IB1AutSwch1 := "STDLog0", IB1FuncBtn1 :=, IB1Serv1 := "STDLog0", IB1SigTest1 := "STDLog0", II_FuncBtn1PanelNr := 11, IB1Ack2 := "STATUS_100+UH11".SF03_14, IB1AckSfty2 := "STATUS_100+UH11".SF04_14, IB1AckSftyReq2 := "JSA0Comm", IB1AutStartBtn2 := "STATUS_100+UH11".SF02_14, IB1ManSwch2 := "STDLog0", IB1AutSwch2 := "STDLog0", IB1FuncBtn2 :=, IB1Serv2 := "STDLog0", IB1SigTest2 := "STDLog0", II_FuncBtn2PanelNr := 2, IB1AckSftyReq3 := "JSA0Comm", IB1ManSwch3 := "STDLog0", IB1AutSwch3 := "STDLog0", IB1FuncBtn3 :=, IB1Serv3 := "STDLog0", IB1SigTest3 := "STDLog0", II_FuncBtn3PanelNr := 3, IB1Rmt := "STDLog1", IB1ClrSel := "JSA0Comm", IB1Req1DevSel := "JSA0Comm", IB1Blink := "STDBlink1,0/1,0", IB1AlmSupp := #TS_Zone.AlarmSuppress, II_DevSelNr := #TS_Zone.DevSelNr, XS_Parameter := "HMI_PARAM_Zone100".Mode, XS_Command := "HMI_CMD_Zone100".Mode, OS_Status => "STATUS_Zone100".Mode, OB1AckFlt1 => #TB1AckFlt1, OB1AckSfty1 => #TB1AckSafety1, OB1AutStart1 => #TB1AutStart1, OB1FuncBtn1 =>, OB1SigAcs1 => #TB1SigAcs1, OB1SigRed1 => #TB1SigRed1, OB1SigYlw1 => #TB1SigYlw1, OB1SigGrn1 => #TB1SigGrn1, OB1AckFlt2 =>, OB1AckSfty2 =>, OB1AutStart2 =>, OB1FuncBtn2 =>, OB1SigAcs2 =>, OB1SigRed2 =>, OB1SigYlw2 =>, OB1SigGrn2 =>, OB1AckFlt3 =>, OB1AckSfty3 =>, OB1AutStart3 =>, OB1FuncBtn3 =>, OB1SigAcs3 =>, OB1SigRed3 =>, OB1SigYlw3 =>, OB1SigGrn3 =>)
   END_RUNG
   RUNG wire#powerrail
      Contact( #TB1ReqEndOfCycle )
   END_RUNG wire#w1
   RUNG wire#powerrail
      Contact( "STATUS_000+UH10".SF03_14 )
   END_RUNG wire#w2
   RUNG wire#powerrail
      Contact( "STATUS_000+UH11".SF03_14 )
   END_RUNG wire#w2
   RUNG wire#powerrail
      Contact( "STATUS_000+UH10".SF04_14 )
   END_RUNG wire#w3
   RUNG wire#powerrail
      Contact( "STATUS_000+UH11".SF04_14 )
   END_RUNG wire#w3
   RUNG wire#powerrail
      Contact( "STATUS_000+UH10".SF02_14 )
   END_RUNG wire#w4
   RUNG wire#powerrail
      Contact( "STATUS_000+UH11".SF02_14 )
   END_RUNG wire#w4
   RUNG wire#powerrail
      Contact( "STATUS_100+UH12".SF03_14 )
   END_RUNG wire#w5
   RUNG wire#powerrail
      Contact( "STATUS_100+UH13".SF03_14 )
   END_RUNG wire#w5
   RUNG wire#powerrail
      Contact( "STATUS_100+UH12".SF04_14 )
   END_RUNG wire#w6
   RUNG wire#powerrail
      Contact( "STATUS_100+UH13".SF04_14 )
   END_RUNG wire#w6
   RUNG wire#powerrail
      Contact( "STATUS_100+UH12".SF02_14 )
   END_RUNG wire#w7
   RUNG wire#powerrail
      Contact( "STATUS_100+UH13".SF02_14 )
   END_RUNG wire#w7
   // the same network as SCL:
   #SF_ZoneMode(IB1SftyOK := #TS_Zone.SafetyOK,   // "STD_Zone"
                IB1CollWrn := #TS_Zone.CollWrn,
                IB1CollErr := #TS_Zone.CollErr,
                IB1AllAutoRun := #TS_Zone.AllInAut,
                IB1AllEndOfCycle := #TS_Zone.AllEndOfCycle,
                IB1AllEndOfProd := #TS_Zone.AllEndOfProd,
                IB1AllInBasePos := #TS_Zone.AllInBasePos,
                IB1AutStartEn := #TS_Zone.StartEn,
                IB1ReqEndOfCycle := #TB1ReqEndOfCycle,
                IB1ReqEndOfProdAct := #TB1ReqEndOfProd,
                IB1ReqEndOfProdCncl := #TS_Zone.AllEndOfProd,
                IB1Ack1 := "STATUS_000+UH10".SF03_14 OR "STATUS_000+UH11".SF03_14,
                IB1AckSfty1 := "STATUS_000+UH10".SF04_14 OR "STATUS_000+UH11".SF04_14,
                IB1AckSftyReq1 := "JSA0Comm",
                IB1AutStartBtn1 := "STATUS_000+UH10".SF02_14 OR "STATUS_000+UH11".SF02_14,
                IB1ManSwch1 := "STDLog0",
                IB1AutSwch1 := "STDLog0",
                IB1Serv1 := "STDLog0",
                IB1SigTest1 := "STDLog0",
                II_FuncBtn1PanelNr := 11,
                IB1Ack2 := "STATUS_100+UH11".SF03_14,
                IB1AckSfty2 := "STATUS_100+UH11".SF04_14,
                IB1AckSftyReq2 := "JSA0Comm",
                IB1AutStartBtn2 := "STATUS_100+UH11".SF02_14,
                IB1ManSwch2 := "STDLog0",
                IB1AutSwch2 := "STDLog0",
                IB1Serv2 := "STDLog0",
                IB1SigTest2 := "STDLog0",
                II_FuncBtn2PanelNr := 2,
                IB1Ack3 := "STATUS_100+UH12".SF03_14 OR "STATUS_100+UH13".SF03_14,
                IB1AckSfty3 := "STATUS_100+UH12".SF04_14 OR "STATUS_100+UH13".SF04_14,
                IB1AckSftyReq3 := "JSA0Comm",
                IB1AutStartBtn3 := "STATUS_100+UH12".SF02_14 OR "STATUS_100+UH13".SF02_14,
                IB1ManSwch3 := "STDLog0",
                IB1AutSwch3 := "STDLog0",
                IB1Serv3 := "STDLog0",
                IB1SigTest3 := "STDLog0",
                II_FuncBtn3PanelNr := 3,
                IB1Rmt := "STDLog1",
                IB1ClrSel := "JSA0Comm",
                IB1Req1DevSel := "JSA0Comm",
                IB1Blink := "STDBlink1,0/1,0",
                IB1AlmSupp := #TS_Zone.AlarmSuppress,
                II_DevSelNr := #TS_Zone.DevSelNr,
                XS_Parameter := "HMI_PARAM_Zone100".Mode,
                XS_Command := "HMI_CMD_Zone100".Mode,
                OS_Status => "STATUS_Zone100".Mode,
                OB1AckFlt1 => #TB1AckFlt1,
                OB1AckSfty1 => #TB1AckSafety1,
                OB1AutStart1 => #TB1AutStart1,
                OB1SigAcs1 => #TB1SigAcs1,
                OB1SigRed1 => #TB1SigRed1,
                OB1SigYlw1 => #TB1SigYlw1,
                OB1SigGrn1 => #TB1SigGrn1);
END_REGION

REGION Network 21: Zone 100 - Signalization
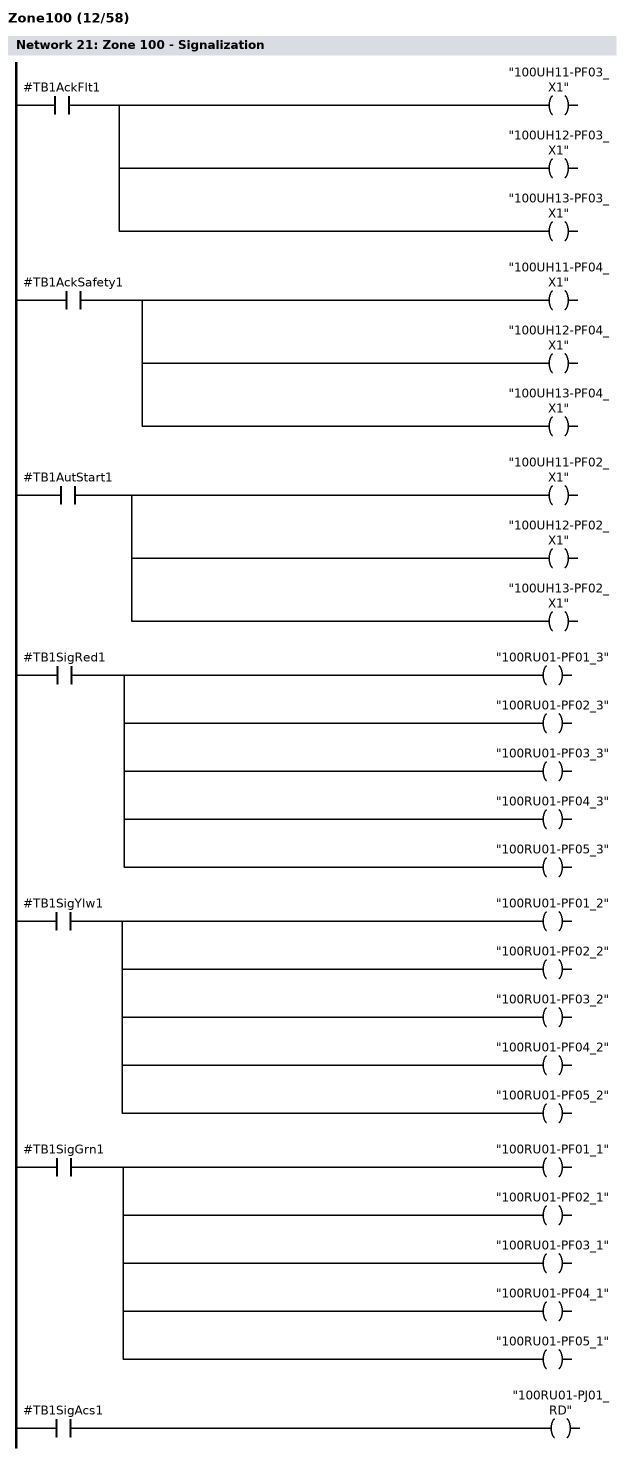
   RUNG wire#powerrail
      Contact( #TB1AckFlt1 )
      wire#w1
      Coil( "100UH11-PF03_X1" )
   END_RUNG
   RUNG wire#w1
      Coil( "100UH12-PF03_X1" )
   END_RUNG
   RUNG wire#w1
      Coil( "100UH13-PF03_X1" )
   END_RUNG
   RUNG wire#powerrail
      Contact( #TB1AckSafety1 )
      wire#w2
      Coil( "100UH11-PF04_X1" )
   END_RUNG
   RUNG wire#w2
      Coil( "100UH12-PF04_X1" )
   END_RUNG
   RUNG wire#w2
      Coil( "100UH13-PF04_X1" )
   END_RUNG
   RUNG wire#powerrail
      Contact( #TB1AutStart1 )
      wire#w3
      Coil( "100UH11-PF02_X1" )
   END_RUNG
   RUNG wire#w3
      Coil( "100UH12-PF02_X1" )
   END_RUNG
   RUNG wire#w3
      Coil( "100UH13-PF02_X1" )
   END_RUNG
   RUNG wire#powerrail
      Contact( #TB1SigRed1 )
      wire#w4
      Coil( "100RU01-PF01_3" )
   END_RUNG
   RUNG wire#w4
      Coil( "100RU01-PF02_3" )
   END_RUNG
   RUNG wire#w4
      Coil( "100RU01-PF03_3" )
   END_RUNG
   RUNG wire#w4
      Coil( "100RU01-PF04_3" )
   END_RUNG
   RUNG wire#w4
      Coil( "100RU01-PF05_3" )
   END_RUNG
   RUNG wire#powerrail
      Contact( #TB1SigYlw1 )
      wire#w5
      Coil( "100RU01-PF01_2" )
   END_RUNG
   RUNG wire#w5
      Coil( "100RU01-PF02_2" )
   END_RUNG
   RUNG wire#w5
      Coil( "100RU01-PF03_2" )
   END_RUNG
   RUNG wire#w5
      Coil( "100RU01-PF04_2" )
   END_RUNG
   RUNG wire#w5
      Coil( "100RU01-PF05_2" )
   END_RUNG
   RUNG wire#powerrail
      Contact( #TB1SigGrn1 )
      wire#w6
      Coil( "100RU01-PF01_1" )
   END_RUNG
   RUNG wire#w6
      Coil( "100RU01-PF02_1" )
   END_RUNG
   RUNG wire#w6
      Coil( "100RU01-PF03_1" )
   END_RUNG
   RUNG wire#w6
      Coil( "100RU01-PF04_1" )
   END_RUNG
   RUNG wire#w6
      Coil( "100RU01-PF05_1" )
   END_RUNG
   RUNG wire#powerrail
      Contact( #TB1SigAcs1 )
      Coil( "100RU01-PJ01_RD" )
   END_RUNG
   // the same network as SCL:
   "100UH11-PF03_X1" := #TB1AckFlt1;
   "100UH12-PF03_X1" := #TB1AckFlt1;
   "100UH13-PF03_X1" := #TB1AckFlt1;
   "100UH11-PF04_X1" := #TB1AckSafety1;
   "100UH12-PF04_X1" := #TB1AckSafety1;
   "100UH13-PF04_X1" := #TB1AckSafety1;
   "100UH11-PF02_X1" := #TB1AutStart1;
   "100UH12-PF02_X1" := #TB1AutStart1;
   "100UH13-PF02_X1" := #TB1AutStart1;
   "100RU01-PF01_3" := #TB1SigRed1;
   "100RU01-PF02_3" := #TB1SigRed1;
   "100RU01-PF03_3" := #TB1SigRed1;
   "100RU01-PF04_3" := #TB1SigRed1;
   "100RU01-PF05_3" := #TB1SigRed1;
   "100RU01-PF01_2" := #TB1SigYlw1;
   "100RU01-PF02_2" := #TB1SigYlw1;
   "100RU01-PF03_2" := #TB1SigYlw1;
   "100RU01-PF04_2" := #TB1SigYlw1;
   "100RU01-PF05_2" := #TB1SigYlw1;
   "100RU01-PF01_1" := #TB1SigGrn1;
   "100RU01-PF02_1" := #TB1SigGrn1;
   "100RU01-PF03_1" := #TB1SigGrn1;
   "100RU01-PF04_1" := #TB1SigGrn1;
   "100RU01-PF05_1" := #TB1SigGrn1;
   "100RU01-PJ01_RD" := #TB1SigAcs1;
END_REGION

REGION Network 22: *************** Station KAS1 ***************
END_REGION

REGION Network 23: Station KAS1 - There is some device that is still running
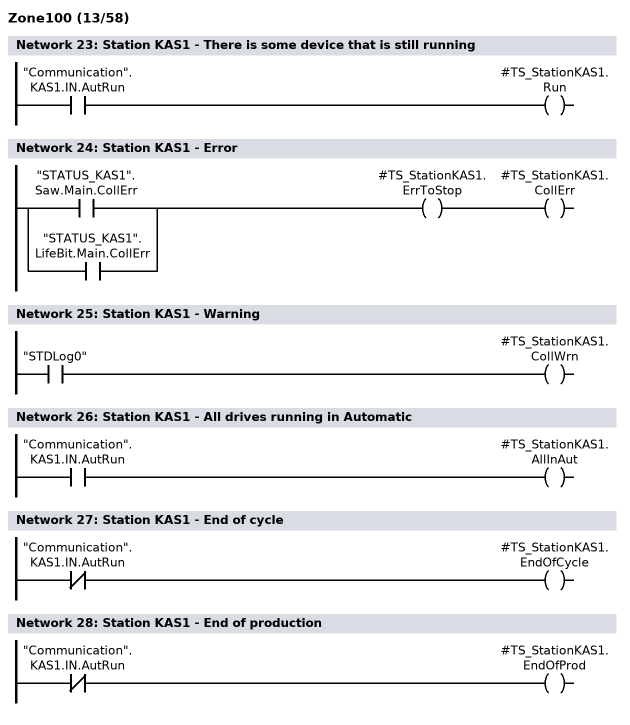
   RUNG wire#powerrail
      Contact( "Communication".KAS1.IN.AutRun )
      Coil( #TS_StationKAS1.Run )
   END_RUNG
   // the same network as SCL:
   #TS_StationKAS1.Run := "Communication".KAS1.IN.AutRun;
END_REGION

REGION Network 24: Station KAS1 - Error
   RUNG wire#powerrail
      Contact( "STATUS_KAS1".Saw.Main.CollErr )
      wire#w1
      Coil( #TS_StationKAS1.ErrToStop )
      Coil( #TS_StationKAS1.CollErr )
   END_RUNG
   RUNG wire#powerrail
      Contact( "STATUS_KAS1".LifeBit.Main.CollErr )
   END_RUNG wire#w1
   // the same network as SCL:
   #TS_StationKAS1.ErrToStop := "STATUS_KAS1".Saw.Main.CollErr OR "STATUS_KAS1".LifeBit.Main.CollErr;
   #TS_StationKAS1.CollErr := #TS_StationKAS1.ErrToStop;
END_REGION

REGION Network 25: Station KAS1 - Warning
   RUNG wire#powerrail
      Contact( "STDLog0" )
      Coil( #TS_StationKAS1.CollWrn )
   END_RUNG
   // the same network as SCL:
   #TS_StationKAS1.CollWrn := "STDLog0";
END_REGION

REGION Network 26: Station KAS1 - All drives running in Automatic
   RUNG wire#powerrail
      Contact( "Communication".KAS1.IN.AutRun )
      Coil( #TS_StationKAS1.AllInAut )
   END_RUNG
   // the same network as SCL:
   #TS_StationKAS1.AllInAut := "Communication".KAS1.IN.AutRun;
END_REGION

REGION Network 27: Station KAS1 - End of cycle
   RUNG wire#powerrail
      I_Contact( "Communication".KAS1.IN.AutRun )
      Coil( #TS_StationKAS1.EndOfCycle )
   END_RUNG
   // the same network as SCL:
   #TS_StationKAS1.EndOfCycle := NOT "Communication".KAS1.IN.AutRun;
END_REGION

REGION Network 28: Station KAS1 - End of production
   RUNG wire#powerrail
      I_Contact( "Communication".KAS1.IN.AutRun )
      Coil( #TS_StationKAS1.EndOfProd )
   END_RUNG
   // the same network as SCL:
   #TS_StationKAS1.EndOfProd := NOT "Communication".KAS1.IN.AutRun;
END_REGION

REGION Network 29: Station KAS1 - Main control
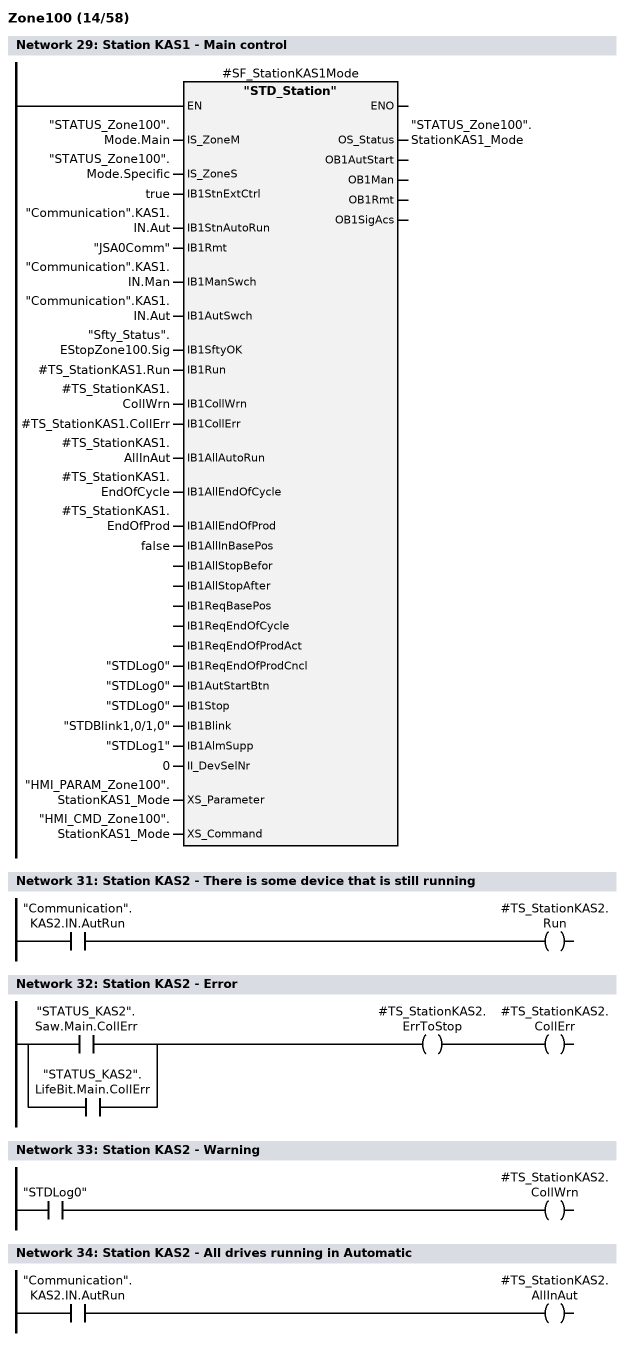
   RUNG wire#powerrail
      #SF_StationKAS1Mode(IS_ZoneM := "STATUS_Zone100".Mode.Main, IS_ZoneS := "STATUS_Zone100".Mode.Specific, IB1StnExtCtrl := true, IB1StnAutoRun := "Communication".KAS1.IN.Aut, IB1Rmt := "JSA0Comm", IB1ManSwch := "Communication".KAS1.IN.Man, IB1AutSwch := "Communication".KAS1.IN.Aut, IB1SftyOK := "Sfty_Status".EStopZone100.Sig, IB1Run := #TS_StationKAS1.Run, IB1CollWrn := #TS_StationKAS1.CollWrn, IB1CollErr := #TS_StationKAS1.CollErr, IB1AllAutoRun := #TS_StationKAS1.AllInAut, IB1AllEndOfCycle := #TS_StationKAS1.EndOfCycle, IB1AllEndOfProd := #TS_StationKAS1.EndOfProd, IB1AllInBasePos := false, IB1AllStopBefor :=, IB1AllStopAfter :=, IB1ReqBasePos :=, IB1ReqEndOfCycle :=, IB1ReqEndOfProdAct :=, IB1ReqEndOfProdCncl := "STDLog0", IB1AutStartBtn := "STDLog0", IB1Stop := "STDLog0", IB1Blink := "STDBlink1,0/1,0", IB1AlmSupp := "STDLog1", II_DevSelNr := 0, XS_Parameter := "HMI_PARAM_Zone100".StationKAS1_Mode, XS_Command := "HMI_CMD_Zone100".StationKAS1_Mode, OS_Status => "STATUS_Zone100".StationKAS1_Mode, OB1AutStart =>, OB1Man =>, OB1Rmt =>, OB1SigAcs =>)
   END_RUNG
   // the same network as SCL:
   #SF_StationKAS1Mode(IS_ZoneM := "STATUS_Zone100".Mode.Main,   // "STD_Station"
                       IS_ZoneS := "STATUS_Zone100".Mode.Specific,
                       IB1StnExtCtrl := true,
                       IB1StnAutoRun := "Communication".KAS1.IN.Aut,
                       IB1Rmt := "JSA0Comm",
                       IB1ManSwch := "Communication".KAS1.IN.Man,
                       IB1AutSwch := "Communication".KAS1.IN.Aut,
                       IB1SftyOK := "Sfty_Status".EStopZone100.Sig,
                       IB1Run := #TS_StationKAS1.Run,
                       IB1CollWrn := #TS_StationKAS1.CollWrn,
                       IB1CollErr := #TS_StationKAS1.CollErr,
                       IB1AllAutoRun := #TS_StationKAS1.AllInAut,
                       IB1AllEndOfCycle := #TS_StationKAS1.EndOfCycle,
                       IB1AllEndOfProd := #TS_StationKAS1.EndOfProd,
                       IB1AllInBasePos := false,
                       IB1ReqEndOfProdCncl := "STDLog0",
                       IB1AutStartBtn := "STDLog0",
                       IB1Stop := "STDLog0",
                       IB1Blink := "STDBlink1,0/1,0",
                       IB1AlmSupp := "STDLog1",
                       II_DevSelNr := 0,
                       XS_Parameter := "HMI_PARAM_Zone100".StationKAS1_Mode,
                       XS_Command := "HMI_CMD_Zone100".StationKAS1_Mode,
                       OS_Status => "STATUS_Zone100".StationKAS1_Mode);
END_REGION

REGION Network 30: *************** Station KAS2 ***************
END_REGION

REGION Network 31: Station KAS2 - There is some device that is still running
   RUNG wire#powerrail
      Contact( "Communication".KAS2.IN.AutRun )
      Coil( #TS_StationKAS2.Run )
   END_RUNG
   // the same network as SCL:
   #TS_StationKAS2.Run := "Communication".KAS2.IN.AutRun;
END_REGION

REGION Network 32: Station KAS2 - Error
   RUNG wire#powerrail
      Contact( "STATUS_KAS2".Saw.Main.CollErr )
      wire#w1
      Coil( #TS_StationKAS2.ErrToStop )
      Coil( #TS_StationKAS2.CollErr )
   END_RUNG
   RUNG wire#powerrail
      Contact( "STATUS_KAS2".LifeBit.Main.CollErr )
   END_RUNG wire#w1
   // the same network as SCL:
   #TS_StationKAS2.ErrToStop := "STATUS_KAS2".Saw.Main.CollErr OR "STATUS_KAS2".LifeBit.Main.CollErr;
   #TS_StationKAS2.CollErr := #TS_StationKAS2.ErrToStop;
END_REGION

REGION Network 33: Station KAS2 - Warning
   RUNG wire#powerrail
      Contact( "STDLog0" )
      Coil( #TS_StationKAS2.CollWrn )
   END_RUNG
   // the same network as SCL:
   #TS_StationKAS2.CollWrn := "STDLog0";
END_REGION

REGION Network 34: Station KAS2 - All drives running in Automatic
   RUNG wire#powerrail
      Contact( "Communication".KAS2.IN.AutRun )
      Coil( #TS_StationKAS2.AllInAut )
   END_RUNG
   // the same network as SCL:
   #TS_StationKAS2.AllInAut := "Communication".KAS2.IN.AutRun;
END_REGION

REGION Network 35: Station KAS2 - End of cycle
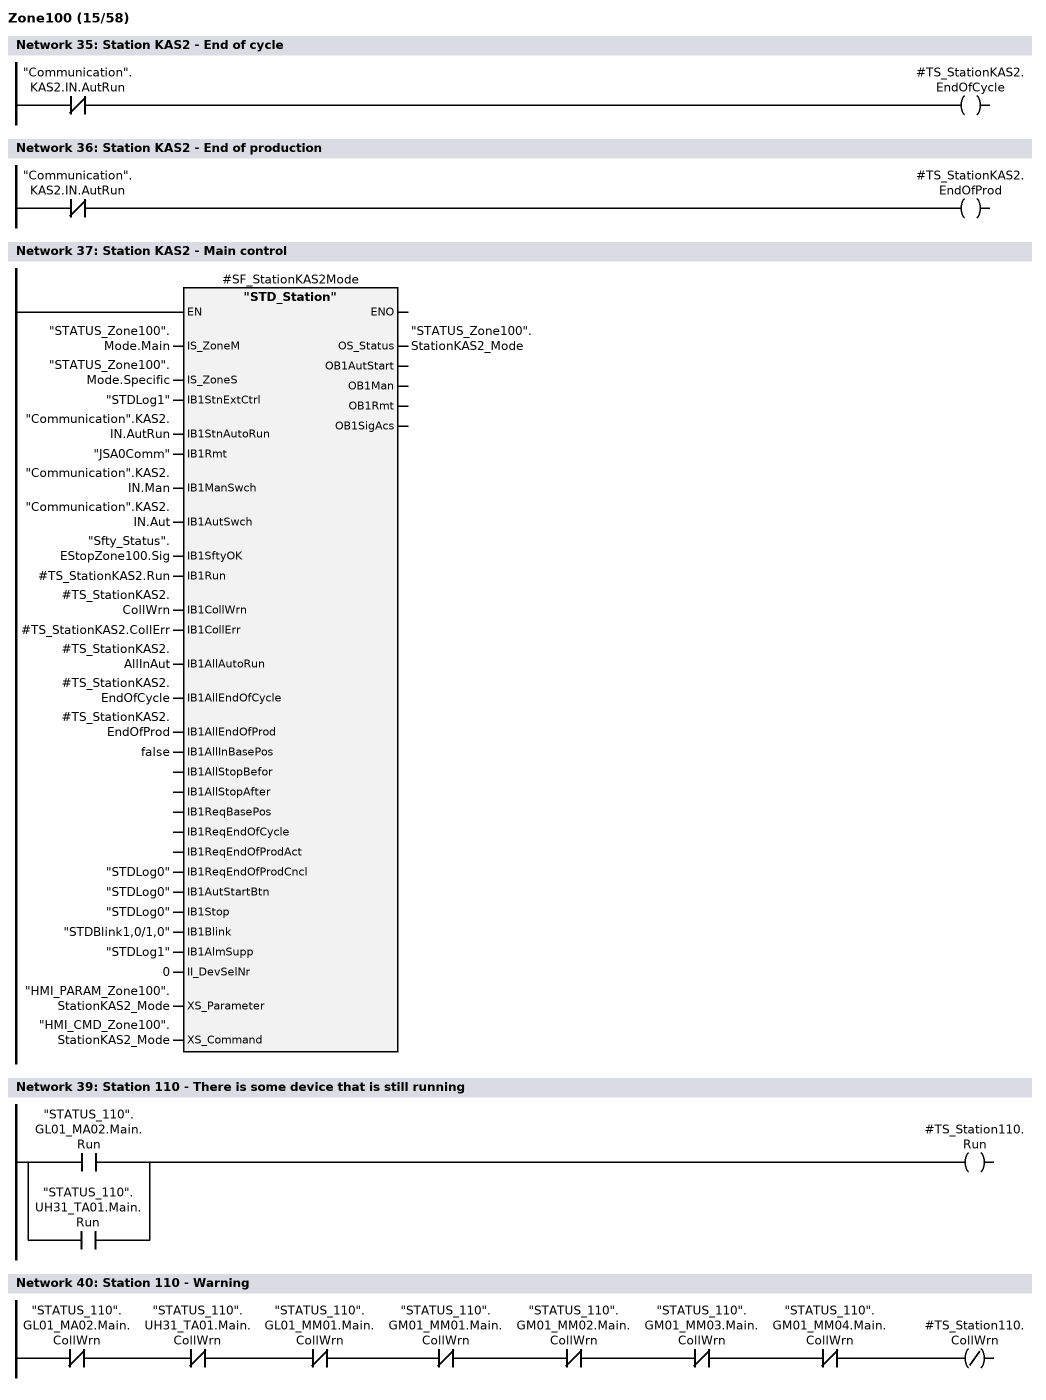
   RUNG wire#powerrail
      I_Contact( "Communication".KAS2.IN.AutRun )
      Coil( #TS_StationKAS2.EndOfCycle )
   END_RUNG
   // the same network as SCL:
   #TS_StationKAS2.EndOfCycle := NOT "Communication".KAS2.IN.AutRun;
END_REGION

REGION Network 36: Station KAS2 - End of production
   RUNG wire#powerrail
      I_Contact( "Communication".KAS2.IN.AutRun )
      Coil( #TS_StationKAS2.EndOfProd )
   END_RUNG
   // the same network as SCL:
   #TS_StationKAS2.EndOfProd := NOT "Communication".KAS2.IN.AutRun;
END_REGION

REGION Network 37: Station KAS2 - Main control
   RUNG wire#powerrail
      #SF_StationKAS2Mode(IS_ZoneM := "STATUS_Zone100".Mode.Main, IS_ZoneS := "STATUS_Zone100".Mode.Specific, IB1StnExtCtrl := "STDLog1", IB1StnAutoRun := "Communication".KAS2.IN.AutRun, IB1Rmt := "JSA0Comm", IB1ManSwch := "Communication".KAS2.IN.Man, IB1AutSwch := "Communication".KAS2.IN.Aut, IB1SftyOK := "Sfty_Status".EStopZone100.Sig, IB1Run := #TS_StationKAS2.Run, IB1CollWrn := #TS_StationKAS2.CollWrn, IB1CollErr := #TS_StationKAS2.CollErr, IB1AllAutoRun := #TS_StationKAS2.AllInAut, IB1AllEndOfCycle := #TS_StationKAS2.EndOfCycle, IB1AllEndOfProd := #TS_StationKAS2.EndOfProd, IB1AllInBasePos := false, IB1AllStopBefor :=, IB1AllStopAfter :=, IB1ReqBasePos :=, IB1ReqEndOfCycle :=, IB1ReqEndOfProdAct :=, IB1ReqEndOfProdCncl := "STDLog0", IB1AutStartBtn := "STDLog0", IB1Stop := "STDLog0", IB1Blink := "STDBlink1,0/1,0", IB1AlmSupp := "STDLog1", II_DevSelNr := 0, XS_Parameter := "HMI_PARAM_Zone100".StationKAS2_Mode, XS_Command := "HMI_CMD_Zone100".StationKAS2_Mode, OS_Status => "STATUS_Zone100".StationKAS2_Mode, OB1AutStart =>, OB1Man =>, OB1Rmt =>, OB1SigAcs =>)
   END_RUNG
   // the same network as SCL:
   #SF_StationKAS2Mode(IS_ZoneM := "STATUS_Zone100".Mode.Main,   // "STD_Station"
                       IS_ZoneS := "STATUS_Zone100".Mode.Specific,
                       IB1StnExtCtrl := "STDLog1",
                       IB1StnAutoRun := "Communication".KAS2.IN.AutRun,
                       IB1Rmt := "JSA0Comm",
                       IB1ManSwch := "Communication".KAS2.IN.Man,
                       IB1AutSwch := "Communication".KAS2.IN.Aut,
                       IB1SftyOK := "Sfty_Status".EStopZone100.Sig,
                       IB1Run := #TS_StationKAS2.Run,
                       IB1CollWrn := #TS_StationKAS2.CollWrn,
                       IB1CollErr := #TS_StationKAS2.CollErr,
                       IB1AllAutoRun := #TS_StationKAS2.AllInAut,
                       IB1AllEndOfCycle := #TS_StationKAS2.EndOfCycle,
                       IB1AllEndOfProd := #TS_StationKAS2.EndOfProd,
                       IB1AllInBasePos := false,
                       IB1ReqEndOfProdCncl := "STDLog0",
                       IB1AutStartBtn := "STDLog0",
                       IB1Stop := "STDLog0",
                       IB1Blink := "STDBlink1,0/1,0",
                       IB1AlmSupp := "STDLog1",
                       II_DevSelNr := 0,
                       XS_Parameter := "HMI_PARAM_Zone100".StationKAS2_Mode,
                       XS_Command := "HMI_CMD_Zone100".StationKAS2_Mode,
                       OS_Status => "STATUS_Zone100".StationKAS2_Mode);
END_REGION

REGION Network 38: *************** Station 110 ***************
END_REGION

REGION Network 39: Station 110 - There is some device that is still running
   RUNG wire#powerrail
      Contact( "STATUS_110".GL01_MA02.Main.Run )
      wire#w1
      Coil( #TS_Station110.Run )
   END_RUNG
   RUNG wire#powerrail
      Contact( "STATUS_110".UH31_TA01.Main.Run )
   END_RUNG wire#w1
   // the same network as SCL:
   #TS_Station110.Run := "STATUS_110".GL01_MA02.Main.Run OR "STATUS_110".UH31_TA01.Main.Run;
END_REGION

REGION Network 40: Station 110 - Warning
   RUNG wire#powerrail
      I_Contact( "STATUS_110".GL01_MA02.Main.CollWrn )
      I_Contact( "STATUS_110".UH31_TA01.Main.CollWrn )
      I_Contact( "STATUS_110".GL01_MM01.Main.CollWrn )
      I_Contact( "STATUS_110".GM01_MM01.Main.CollWrn )
      I_Contact( "STATUS_110".GM01_MM02.Main.CollWrn )
      I_Contact( "STATUS_110".GM01_MM03.Main.CollWrn )
      I_Contact( "STATUS_110".GM01_MM04.Main.CollWrn )
      I_Coil( #TS_Station110.CollWrn )
   END_RUNG
   // the same network as SCL:
   #TS_Station110.CollWrn := NOT (NOT "STATUS_110".GL01_MA02.Main.CollWrn AND NOT "STATUS_110".UH31_TA01.Main.CollWrn AND NOT "STATUS_110".GL01_MM01.Main.CollWrn AND NOT "STATUS_110".GM01_MM01.Main.CollWrn AND NOT "STATUS_110".GM01_MM02.Main.CollWrn AND NOT "STATUS_110".GM01_MM03.Main.CollWrn AND NOT "STATUS_110".GM01_MM04.Main.CollWrn);
END_REGION

REGION Network 41: Station 110 - Error to stop
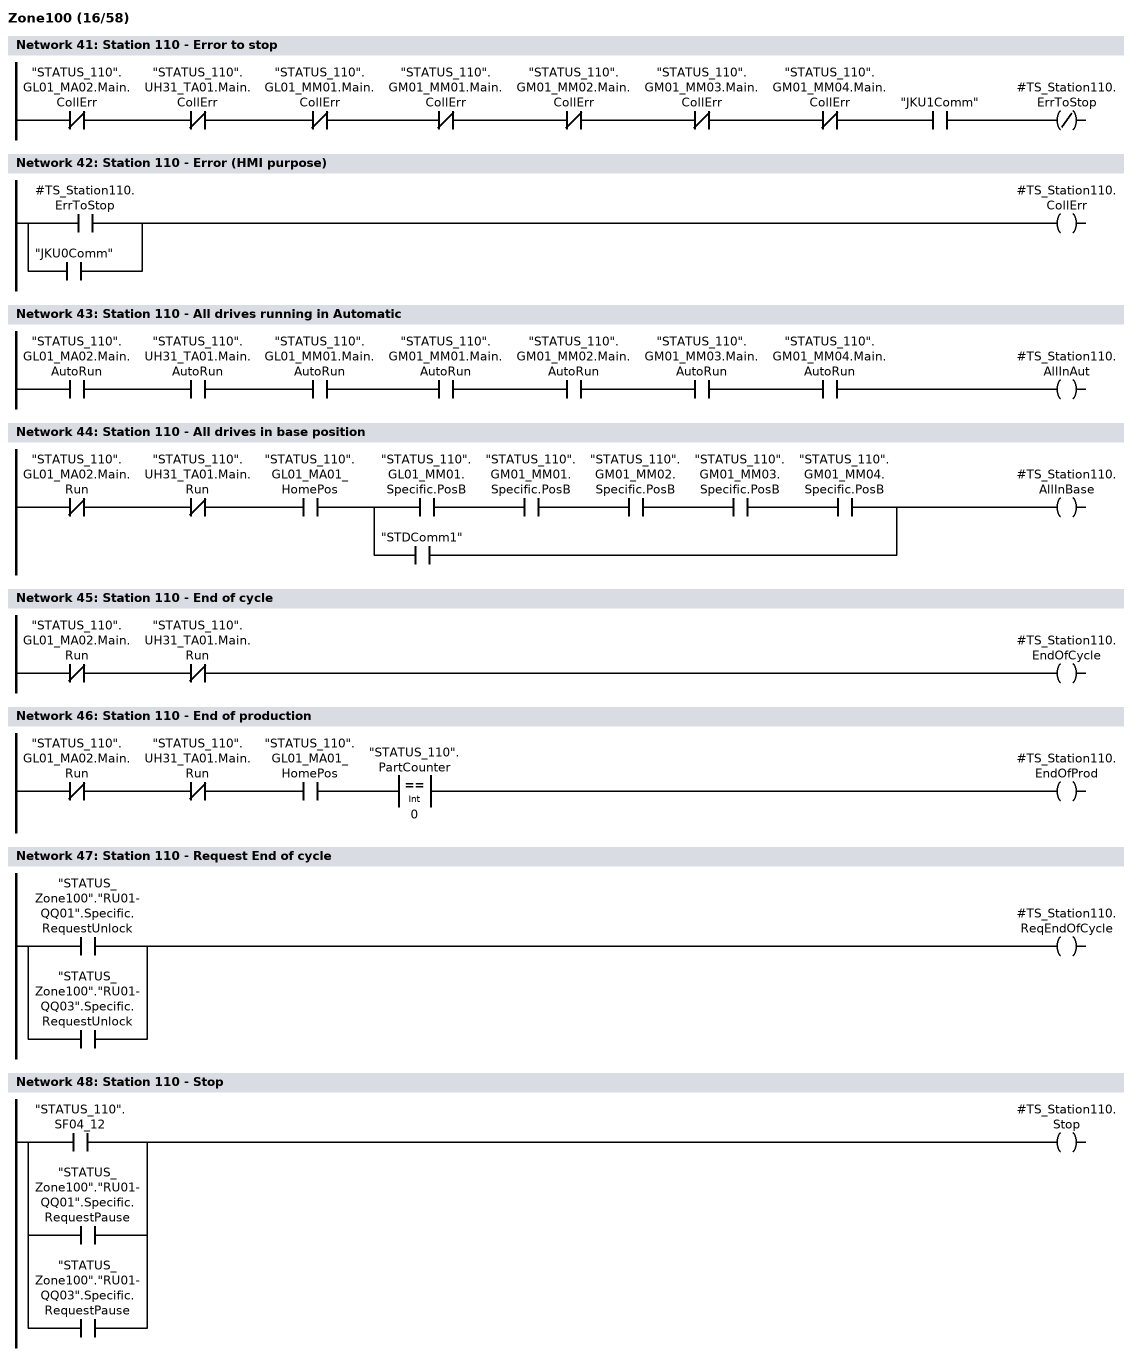
   RUNG wire#powerrail
      I_Contact( "STATUS_110".GL01_MA02.Main.CollErr )
      I_Contact( "STATUS_110".UH31_TA01.Main.CollErr )
      I_Contact( "STATUS_110".GL01_MM01.Main.CollErr )
      I_Contact( "STATUS_110".GM01_MM01.Main.CollErr )
      I_Contact( "STATUS_110".GM01_MM02.Main.CollErr )
      I_Contact( "STATUS_110".GM01_MM03.Main.CollErr )
      I_Contact( "STATUS_110".GM01_MM04.Main.CollErr )
      Contact( "JKU1Comm" )
      I_Coil( #TS_Station110.ErrToStop )
   END_RUNG
   // the same network as SCL:
   #TS_Station110.ErrToStop := NOT (NOT "STATUS_110".GL01_MA02.Main.CollErr AND NOT "STATUS_110".UH31_TA01.Main.CollErr AND NOT "STATUS_110".GL01_MM01.Main.CollErr AND NOT "STATUS_110".GM01_MM01.Main.CollErr AND NOT "STATUS_110".GM01_MM02.Main.CollErr AND NOT "STATUS_110".GM01_MM03.Main.CollErr AND NOT "STATUS_110".GM01_MM04.Main.CollErr AND "JKU1Comm");
END_REGION

REGION Network 42: Station 110 - Error (HMI purpose)
   RUNG wire#powerrail
      Contact( #TS_Station110.ErrToStop )
      wire#w1
      Coil( #TS_Station110.CollErr )
   END_RUNG
   RUNG wire#powerrail
      Contact( "JKU0Comm" )
   END_RUNG wire#w1
   // the same network as SCL:
   #TS_Station110.CollErr := #TS_Station110.ErrToStop OR "JKU0Comm";
END_REGION

REGION Network 43: Station 110 - All drives running in Automatic
   RUNG wire#powerrail
      Contact( "STATUS_110".GL01_MA02.Main.AutoRun )
      Contact( "STATUS_110".UH31_TA01.Main.AutoRun )
      Contact( "STATUS_110".GL01_MM01.Main.AutoRun )
      Contact( "STATUS_110".GM01_MM01.Main.AutoRun )
      Contact( "STATUS_110".GM01_MM02.Main.AutoRun )
      Contact( "STATUS_110".GM01_MM03.Main.AutoRun )
      Contact( "STATUS_110".GM01_MM04.Main.AutoRun )
      Coil( #TS_Station110.AllInAut )
   END_RUNG
   // the same network as SCL:
   #TS_Station110.AllInAut := "STATUS_110".GL01_MA02.Main.AutoRun AND "STATUS_110".UH31_TA01.Main.AutoRun AND "STATUS_110".GL01_MM01.Main.AutoRun AND "STATUS_110".GM01_MM01.Main.AutoRun AND "STATUS_110".GM01_MM02.Main.AutoRun AND "STATUS_110".GM01_MM03.Main.AutoRun AND "STATUS_110".GM01_MM04.Main.AutoRun;
END_REGION

REGION Network 44: Station 110 - All drives in base position
   RUNG wire#powerrail
      I_Contact( "STATUS_110".GL01_MA02.Main.Run )
      I_Contact( "STATUS_110".UH31_TA01.Main.Run )
      Contact( "STATUS_110".GL01_MA01_HomePos )
      wire#w1
      Contact( "STATUS_110".GL01_MM01.Specific.PosB )
      Contact( "STATUS_110".GM01_MM01.Specific.PosB )
      Contact( "STATUS_110".GM01_MM02.Specific.PosB )
      Contact( "STATUS_110".GM01_MM03.Specific.PosB )
      Contact( "STATUS_110".GM01_MM04.Specific.PosB )
      wire#w2
      Coil( #TS_Station110.AllInBase )
   END_RUNG
   RUNG wire#w1
      Contact( "STDComm1" )
   END_RUNG wire#w2
   // the same network as SCL:
   #TS_Station110.AllInBase := NOT "STATUS_110".GL01_MA02.Main.Run AND NOT "STATUS_110".UH31_TA01.Main.Run AND "STATUS_110".GL01_MA01_HomePos AND (("STATUS_110".GL01_MM01.Specific.PosB AND "STATUS_110".GM01_MM01.Specific.PosB AND "STATUS_110".GM01_MM02.Specific.PosB AND "STATUS_110".GM01_MM03.Specific.PosB AND "STATUS_110".GM01_MM04.Specific.PosB) OR "STDComm1");
END_REGION

REGION Network 45: Station 110 - End of cycle
   RUNG wire#powerrail
      I_Contact( "STATUS_110".GL01_MA02.Main.Run )
      I_Contact( "STATUS_110".UH31_TA01.Main.Run )
      Coil( #TS_Station110.EndOfCycle )
   END_RUNG
   // the same network as SCL:
   #TS_Station110.EndOfCycle := NOT "STATUS_110".GL01_MA02.Main.Run AND NOT "STATUS_110".UH31_TA01.Main.Run;
END_REGION

REGION Network 46: Station 110 - End of production
   RUNG wire#powerrail
      I_Contact( "STATUS_110".GL01_MA02.Main.Run )
      I_Contact( "STATUS_110".UH31_TA01.Main.Run )
      Contact( "STATUS_110".GL01_MA01_HomePos )
      { S7_Templates := "SrcType := Int" } EQ_Contact(in1 := "STATUS_110".PartCounter, in2 := 0)
      Coil( #TS_Station110.EndOfProd )
   END_RUNG
   // the same network as SCL:
   #TS_Station110.EndOfProd := NOT "STATUS_110".GL01_MA02.Main.Run AND NOT "STATUS_110".UH31_TA01.Main.Run AND "STATUS_110".GL01_MA01_HomePos AND ("STATUS_110".PartCounter = 0);
END_REGION

REGION Network 47: Station 110 - Request End of cycle
   RUNG wire#powerrail
      Contact( "STATUS_Zone100"."RU01-QQ01".Specific.RequestUnlock )
      wire#w1
      Coil( #TS_Station110.ReqEndOfCycle )
   END_RUNG
   RUNG wire#powerrail
      Contact( "STATUS_Zone100"."RU01-QQ03".Specific.RequestUnlock )
   END_RUNG wire#w1
   // the same network as SCL:
   #TS_Station110.ReqEndOfCycle := "STATUS_Zone100"."RU01-QQ01".Specific.RequestUnlock OR "STATUS_Zone100"."RU01-QQ03".Specific.RequestUnlock;
END_REGION

REGION Network 48: Station 110 - Stop
   RUNG wire#powerrail
      Contact( "STATUS_110".SF04_12 )
      wire#w1
      Coil( #TS_Station110.Stop )
   END_RUNG
   RUNG wire#powerrail
      Contact( "STATUS_Zone100"."RU01-QQ01".Specific.RequestPause )
   END_RUNG wire#w1
   RUNG wire#powerrail
      Contact( "STATUS_Zone100"."RU01-QQ03".Specific.RequestPause )
   END_RUNG wire#w1
   // the same network as SCL:
   #TS_Station110.Stop := "STATUS_110".SF04_12 OR "STATUS_Zone100"."RU01-QQ01".Specific.RequestPause OR "STATUS_Zone100"."RU01-QQ03".Specific.RequestPause;
END_REGION

REGION Network 49: Station 110 - Number of selected devices
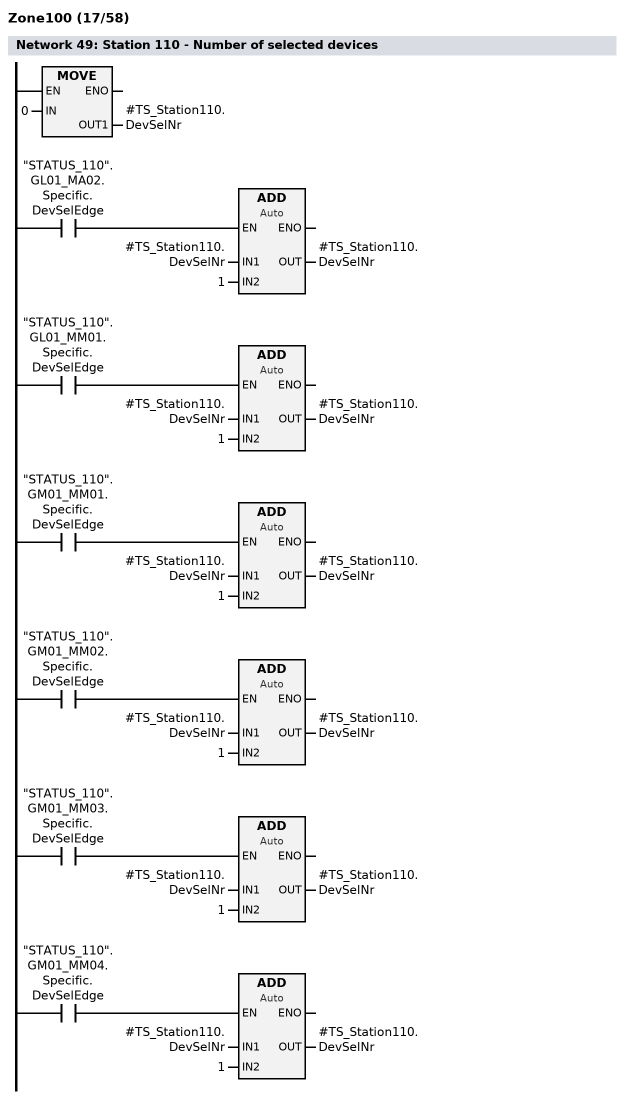
   RUNG wire#powerrail
      Move(in := 0, out1 => #TS_Station110.DevSelNr)
   END_RUNG
   RUNG wire#powerrail
      Contact( "STATUS_110".GL01_MA02.Specific.DevSelEdge )
      Add(in1 := #TS_Station110.DevSelNr, in2 := 1, out => #TS_Station110.DevSelNr)
   END_RUNG
   RUNG wire#powerrail
      Contact( "STATUS_110".GL01_MM01.Specific.DevSelEdge )
      Add(in1 := #TS_Station110.DevSelNr, in2 := 1, out => #TS_Station110.DevSelNr)
   END_RUNG
   RUNG wire#powerrail
      Contact( "STATUS_110".GM01_MM01.Specific.DevSelEdge )
      Add(in1 := #TS_Station110.DevSelNr, in2 := 1, out => #TS_Station110.DevSelNr)
   END_RUNG
   RUNG wire#powerrail
      Contact( "STATUS_110".GM01_MM02.Specific.DevSelEdge )
      Add(in1 := #TS_Station110.DevSelNr, in2 := 1, out => #TS_Station110.DevSelNr)
   END_RUNG
   RUNG wire#powerrail
      Contact( "STATUS_110".GM01_MM03.Specific.DevSelEdge )
      Add(in1 := #TS_Station110.DevSelNr, in2 := 1, out => #TS_Station110.DevSelNr)
   END_RUNG
   RUNG wire#powerrail
      Contact( "STATUS_110".GM01_MM04.Specific.DevSelEdge )
      Add(in1 := #TS_Station110.DevSelNr, in2 := 1, out => #TS_Station110.DevSelNr)
   END_RUNG
   // the same network as SCL:
   #TS_Station110.DevSelNr := 0;
   IF "STATUS_110".GL01_MA02.Specific.DevSelEdge THEN
       #TS_Station110.DevSelNr := #TS_Station110.DevSelNr + 1;
   END_IF;
   IF "STATUS_110".GL01_MM01.Specific.DevSelEdge THEN
       #TS_Station110.DevSelNr := #TS_Station110.DevSelNr + 1;
   END_IF;
   IF "STATUS_110".GM01_MM01.Specific.DevSelEdge THEN
       #TS_Station110.DevSelNr := #TS_Station110.DevSelNr + 1;
   END_IF;
   IF "STATUS_110".GM01_MM02.Specific.DevSelEdge THEN
       #TS_Station110.DevSelNr := #TS_Station110.DevSelNr + 1;
   END_IF;
   IF "STATUS_110".GM01_MM03.Specific.DevSelEdge THEN
       #TS_Station110.DevSelNr := #TS_Station110.DevSelNr + 1;
   END_IF;
   IF "STATUS_110".GM01_MM04.Specific.DevSelEdge THEN
       #TS_Station110.DevSelNr := #TS_Station110.DevSelNr + 1;
   END_IF;
END_REGION

REGION Network 50: Station 110 - Main control
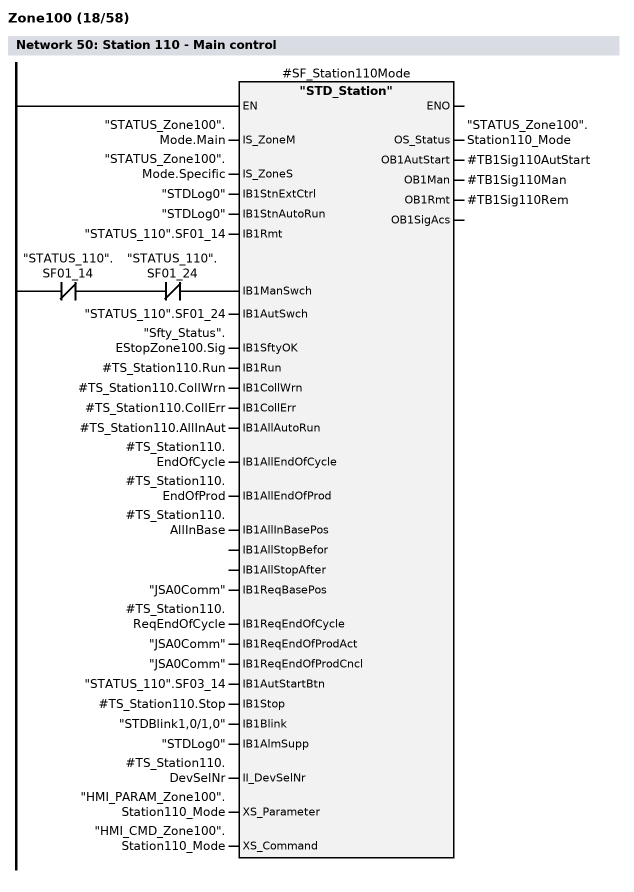
   RUNG wire#powerrail
      #SF_Station110Mode(IB1ManSwch := wire#w1, IS_ZoneM := "STATUS_Zone100".Mode.Main, IS_ZoneS := "STATUS_Zone100".Mode.Specific, IB1StnExtCtrl := "STDLog0", IB1StnAutoRun := "STDLog0", IB1Rmt := "STATUS_110".SF01_14, IB1AutSwch := "STATUS_110".SF01_24, IB1SftyOK := "Sfty_Status".EStopZone100.Sig, IB1Run := #TS_Station110.Run, IB1CollWrn := #TS_Station110.CollWrn, IB1CollErr := #TS_Station110.CollErr, IB1AllAutoRun := #TS_Station110.AllInAut, IB1AllEndOfCycle := #TS_Station110.EndOfCycle, IB1AllEndOfProd := #TS_Station110.EndOfProd, IB1AllInBasePos := #TS_Station110.AllInBase, IB1AllStopBefor :=, IB1AllStopAfter :=, IB1ReqBasePos := "JSA0Comm", IB1ReqEndOfCycle := #TS_Station110.ReqEndOfCycle, IB1ReqEndOfProdAct := "JSA0Comm", IB1ReqEndOfProdCncl := "JSA0Comm", IB1AutStartBtn := "STATUS_110".SF03_14, IB1Stop := #TS_Station110.Stop, IB1Blink := "STDBlink1,0/1,0", IB1AlmSupp := "STDLog0", II_DevSelNr := #TS_Station110.DevSelNr, XS_Parameter := "HMI_PARAM_Zone100".Station110_Mode, XS_Command := "HMI_CMD_Zone100".Station110_Mode, OS_Status => "STATUS_Zone100".Station110_Mode, OB1AutStart => #TB1Sig110AutStart, OB1Man => #TB1Sig110Man, OB1Rmt => #TB1Sig110Rem, OB1SigAcs =>)
   END_RUNG
   RUNG wire#powerrail
      I_Contact( "STATUS_110".SF01_14 )
      I_Contact( "STATUS_110".SF01_24 )
   END_RUNG wire#w1
   // the same network as SCL:
   #SF_Station110Mode(IS_ZoneM := "STATUS_Zone100".Mode.Main,   // "STD_Station"
                      IS_ZoneS := "STATUS_Zone100".Mode.Specific,
                      IB1StnExtCtrl := "STDLog0",
                      IB1StnAutoRun := "STDLog0",
                      IB1Rmt := "STATUS_110".SF01_14,
                      IB1ManSwch := NOT "STATUS_110".SF01_14 AND NOT "STATUS_110".SF01_24,
                      IB1AutSwch := "STATUS_110".SF01_24,
                      IB1SftyOK := "Sfty_Status".EStopZone100.Sig,
                      IB1Run := #TS_Station110.Run,
                      IB1CollWrn := #TS_Station110.CollWrn,
                      IB1CollErr := #TS_Station110.CollErr,
                      IB1AllAutoRun := #TS_Station110.AllInAut,
                      IB1AllEndOfCycle := #TS_Station110.EndOfCycle,
                      IB1AllEndOfProd := #TS_Station110.EndOfProd,
                      IB1AllInBasePos := #TS_Station110.AllInBase,
                      IB1ReqBasePos := "JSA0Comm",
                      IB1ReqEndOfCycle := #TS_Station110.ReqEndOfCycle,
                      IB1ReqEndOfProdAct := "JSA0Comm",
                      IB1ReqEndOfProdCncl := "JSA0Comm",
                      IB1AutStartBtn := "STATUS_110".SF03_14,
                      IB1Stop := #TS_Station110.Stop,
                      IB1Blink := "STDBlink1,0/1,0",
                      IB1AlmSupp := "STDLog0",
                      II_DevSelNr := #TS_Station110.DevSelNr,
                      XS_Parameter := "HMI_PARAM_Zone100".Station110_Mode,
                      XS_Command := "HMI_CMD_Zone100".Station110_Mode,
                      OS_Status => "STATUS_Zone100".Station110_Mode,
                      OB1AutStart => #TB1Sig110AutStart,
                      OB1Man => #TB1Sig110Man,
                      OB1Rmt => #TB1Sig110Rem);
END_REGION

REGION Network 51: Station 110 - Signalization (panel UH11)
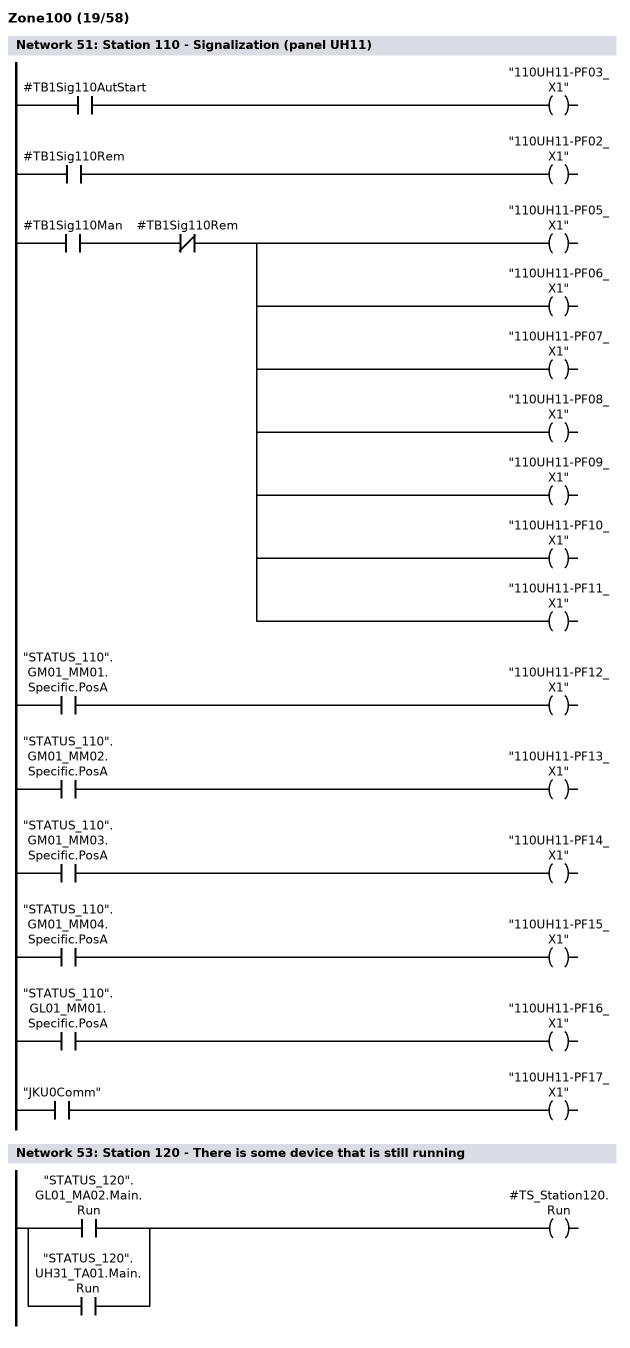
   RUNG wire#powerrail
      Contact( #TB1Sig110AutStart )
      Coil( "110UH11-PF03_X1" )
   END_RUNG
   RUNG wire#powerrail
      Contact( #TB1Sig110Rem )
      Coil( "110UH11-PF02_X1" )
   END_RUNG
   RUNG wire#powerrail
      Contact( #TB1Sig110Man )
      I_Contact( #TB1Sig110Rem )
      wire#w1
      Coil( "110UH11-PF05_X1" )
   END_RUNG
   RUNG wire#w1
      Coil( "110UH11-PF06_X1" )
   END_RUNG
   RUNG wire#w1
      Coil( "110UH11-PF07_X1" )
   END_RUNG
   RUNG wire#w1
      Coil( "110UH11-PF08_X1" )
   END_RUNG
   RUNG wire#w1
      Coil( "110UH11-PF09_X1" )
   END_RUNG
   RUNG wire#w1
      Coil( "110UH11-PF10_X1" )
   END_RUNG
   RUNG wire#w1
      Coil( "110UH11-PF11_X1" )
   END_RUNG
   RUNG wire#powerrail
      Contact( "STATUS_110".GM01_MM01.Specific.PosA )
      Coil( "110UH11-PF12_X1" )
   END_RUNG
   RUNG wire#powerrail
      Contact( "STATUS_110".GM01_MM02.Specific.PosA )
      Coil( "110UH11-PF13_X1" )
   END_RUNG
   RUNG wire#powerrail
      Contact( "STATUS_110".GM01_MM03.Specific.PosA )
      Coil( "110UH11-PF14_X1" )
   END_RUNG
   RUNG wire#powerrail
      Contact( "STATUS_110".GM01_MM04.Specific.PosA )
      Coil( "110UH11-PF15_X1" )
   END_RUNG
   RUNG wire#powerrail
      Contact( "STATUS_110".GL01_MM01.Specific.PosA )
      Coil( "110UH11-PF16_X1" )
   END_RUNG
   RUNG wire#powerrail
      Contact( "JKU0Comm" )
      Coil( "110UH11-PF17_X1" )
   END_RUNG
   // the same network as SCL:
   "110UH11-PF03_X1" := #TB1Sig110AutStart;
   "110UH11-PF02_X1" := #TB1Sig110Rem;
   "110UH11-PF05_X1" := #TB1Sig110Man AND NOT #TB1Sig110Rem;
   "110UH11-PF06_X1" := "110UH11-PF05_X1";
   "110UH11-PF07_X1" := "110UH11-PF05_X1";
   "110UH11-PF08_X1" := "110UH11-PF05_X1";
   "110UH11-PF09_X1" := "110UH11-PF05_X1";
   "110UH11-PF10_X1" := "110UH11-PF05_X1";
   "110UH11-PF11_X1" := "110UH11-PF05_X1";
   "110UH11-PF12_X1" := "STATUS_110".GM01_MM01.Specific.PosA;
   "110UH11-PF13_X1" := "STATUS_110".GM01_MM02.Specific.PosA;
   "110UH11-PF14_X1" := "STATUS_110".GM01_MM03.Specific.PosA;
   "110UH11-PF15_X1" := "STATUS_110".GM01_MM04.Specific.PosA;
   "110UH11-PF16_X1" := "STATUS_110".GL01_MM01.Specific.PosA;
   "110UH11-PF17_X1" := "JKU0Comm";
END_REGION

REGION Network 52: *************** Station 120 ***************
END_REGION

REGION Network 53: Station 120 - There is some device that is still running
   RUNG wire#powerrail
      Contact( "STATUS_120".GL01_MA02.Main.Run )
      wire#w1
      Coil( #TS_Station120.Run )
   END_RUNG
   RUNG wire#powerrail
      Contact( "STATUS_120".UH31_TA01.Main.Run )
   END_RUNG wire#w1
   // the same network as SCL:
   #TS_Station120.Run := "STATUS_120".GL01_MA02.Main.Run OR "STATUS_120".UH31_TA01.Main.Run;
END_REGION

REGION Network 54: Station 120 - Warning
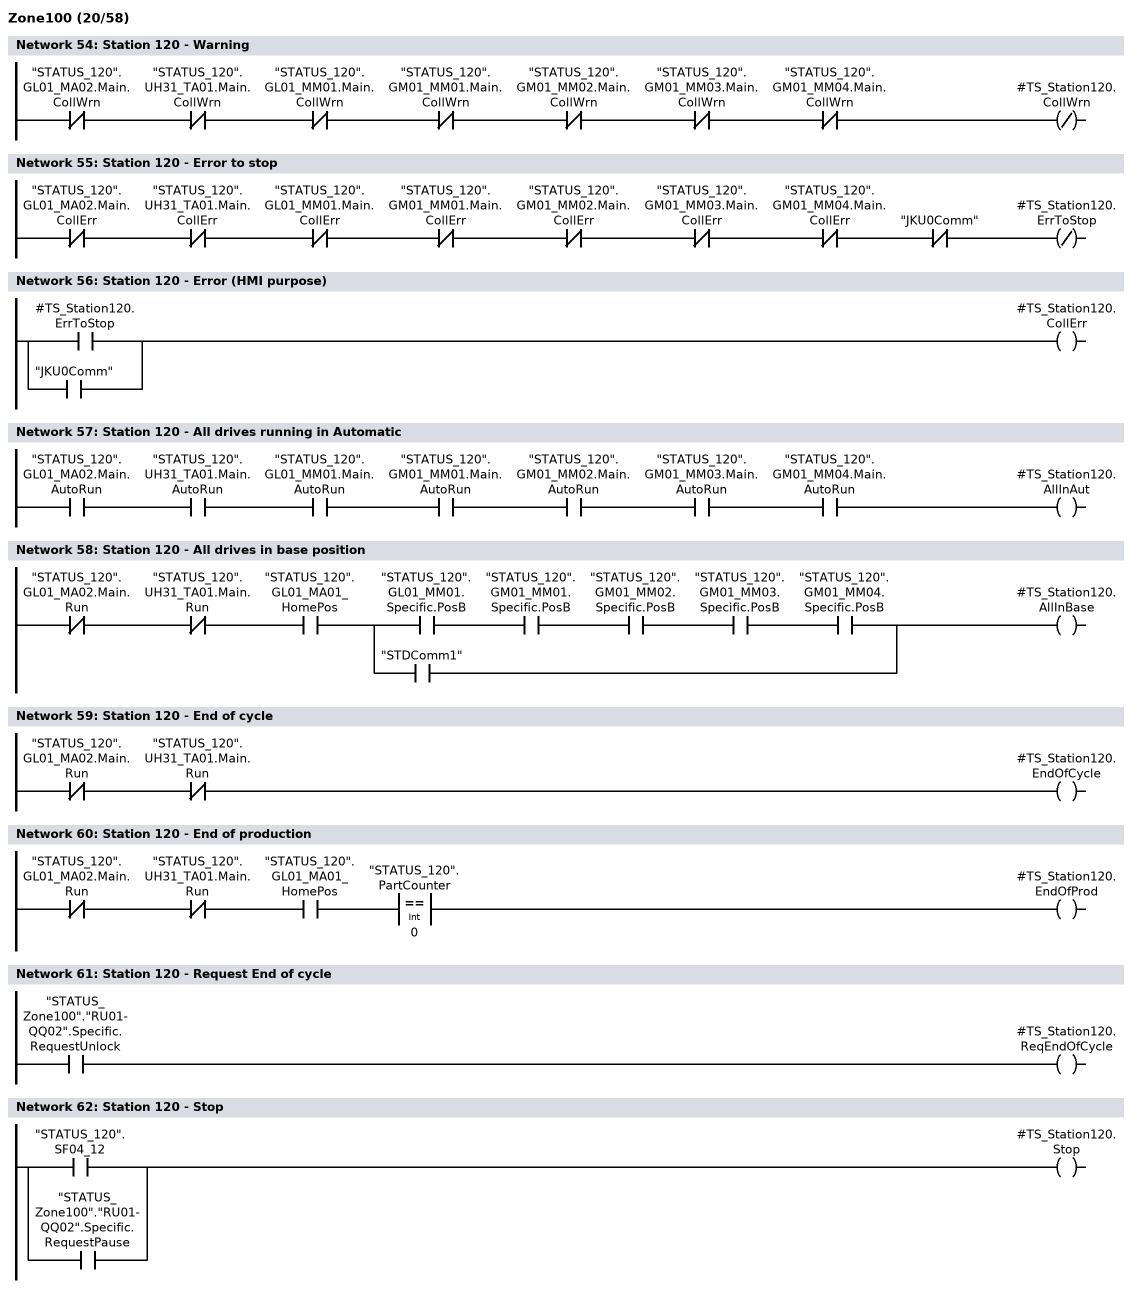
   RUNG wire#powerrail
      I_Contact( "STATUS_120".GL01_MA02.Main.CollWrn )
      I_Contact( "STATUS_120".UH31_TA01.Main.CollWrn )
      I_Contact( "STATUS_120".GL01_MM01.Main.CollWrn )
      I_Contact( "STATUS_120".GM01_MM01.Main.CollWrn )
      I_Contact( "STATUS_120".GM01_MM02.Main.CollWrn )
      I_Contact( "STATUS_120".GM01_MM03.Main.CollWrn )
      I_Contact( "STATUS_120".GM01_MM04.Main.CollWrn )
      I_Coil( #TS_Station120.CollWrn )
   END_RUNG
   // the same network as SCL:
   #TS_Station120.CollWrn := NOT (NOT "STATUS_120".GL01_MA02.Main.CollWrn AND NOT "STATUS_120".UH31_TA01.Main.CollWrn AND NOT "STATUS_120".GL01_MM01.Main.CollWrn AND NOT "STATUS_120".GM01_MM01.Main.CollWrn AND NOT "STATUS_120".GM01_MM02.Main.CollWrn AND NOT "STATUS_120".GM01_MM03.Main.CollWrn AND NOT "STATUS_120".GM01_MM04.Main.CollWrn);
END_REGION

REGION Network 55: Station 120 - Error to stop
   RUNG wire#powerrail
      I_Contact( "STATUS_120".GL01_MA02.Main.CollErr )
      I_Contact( "STATUS_120".UH31_TA01.Main.CollErr )
      I_Contact( "STATUS_120".GL01_MM01.Main.CollErr )
      I_Contact( "STATUS_120".GM01_MM01.Main.CollErr )
      I_Contact( "STATUS_120".GM01_MM02.Main.CollErr )
      I_Contact( "STATUS_120".GM01_MM03.Main.CollErr )
      I_Contact( "STATUS_120".GM01_MM04.Main.CollErr )
      I_Contact( "JKU0Comm" )
      I_Coil( #TS_Station120.ErrToStop )
   END_RUNG
   // the same network as SCL:
   #TS_Station120.ErrToStop := NOT (NOT "STATUS_120".GL01_MA02.Main.CollErr AND NOT "STATUS_120".UH31_TA01.Main.CollErr AND NOT "STATUS_120".GL01_MM01.Main.CollErr AND NOT "STATUS_120".GM01_MM01.Main.CollErr AND NOT "STATUS_120".GM01_MM02.Main.CollErr AND NOT "STATUS_120".GM01_MM03.Main.CollErr AND NOT "STATUS_120".GM01_MM04.Main.CollErr AND NOT "JKU0Comm");
END_REGION

REGION Network 56: Station 120 - Error (HMI purpose)
   RUNG wire#powerrail
      Contact( #TS_Station120.ErrToStop )
      wire#w1
      Coil( #TS_Station120.CollErr )
   END_RUNG
   RUNG wire#powerrail
      Contact( "JKU0Comm" )
   END_RUNG wire#w1
   // the same network as SCL:
   #TS_Station120.CollErr := #TS_Station120.ErrToStop OR "JKU0Comm";
END_REGION

REGION Network 57: Station 120 - All drives running in Automatic
   RUNG wire#powerrail
      Contact( "STATUS_120".GL01_MA02.Main.AutoRun )
      Contact( "STATUS_120".UH31_TA01.Main.AutoRun )
      Contact( "STATUS_120".GL01_MM01.Main.AutoRun )
      Contact( "STATUS_120".GM01_MM01.Main.AutoRun )
      Contact( "STATUS_120".GM01_MM02.Main.AutoRun )
      Contact( "STATUS_120".GM01_MM03.Main.AutoRun )
      Contact( "STATUS_120".GM01_MM04.Main.AutoRun )
      Coil( #TS_Station120.AllInAut )
   END_RUNG
   // the same network as SCL:
   #TS_Station120.AllInAut := "STATUS_120".GL01_MA02.Main.AutoRun AND "STATUS_120".UH31_TA01.Main.AutoRun AND "STATUS_120".GL01_MM01.Main.AutoRun AND "STATUS_120".GM01_MM01.Main.AutoRun AND "STATUS_120".GM01_MM02.Main.AutoRun AND "STATUS_120".GM01_MM03.Main.AutoRun AND "STATUS_120".GM01_MM04.Main.AutoRun;
END_REGION

REGION Network 58: Station 120 - All drives in base position
   RUNG wire#powerrail
      I_Contact( "STATUS_120".GL01_MA02.Main.Run )
      I_Contact( "STATUS_120".UH31_TA01.Main.Run )
      Contact( "STATUS_120".GL01_MA01_HomePos )
      wire#w1
      Contact( "STATUS_120".GL01_MM01.Specific.PosB )
      Contact( "STATUS_120".GM01_MM01.Specific.PosB )
      Contact( "STATUS_120".GM01_MM02.Specific.PosB )
      Contact( "STATUS_120".GM01_MM03.Specific.PosB )
      Contact( "STATUS_120".GM01_MM04.Specific.PosB )
      wire#w2
      Coil( #TS_Station120.AllInBase )
   END_RUNG
   RUNG wire#w1
      Contact( "STDComm1" )
   END_RUNG wire#w2
   // the same network as SCL:
   #TS_Station120.AllInBase := NOT "STATUS_120".GL01_MA02.Main.Run AND NOT "STATUS_120".UH31_TA01.Main.Run AND "STATUS_120".GL01_MA01_HomePos AND (("STATUS_120".GL01_MM01.Specific.PosB AND "STATUS_120".GM01_MM01.Specific.PosB AND "STATUS_120".GM01_MM02.Specific.PosB AND "STATUS_120".GM01_MM03.Specific.PosB AND "STATUS_120".GM01_MM04.Specific.PosB) OR "STDComm1");
END_REGION

REGION Network 59: Station 120 - End of cycle
   RUNG wire#powerrail
      I_Contact( "STATUS_120".GL01_MA02.Main.Run )
      I_Contact( "STATUS_120".UH31_TA01.Main.Run )
      Coil( #TS_Station120.EndOfCycle )
   END_RUNG
   // the same network as SCL:
   #TS_Station120.EndOfCycle := NOT "STATUS_120".GL01_MA02.Main.Run AND NOT "STATUS_120".UH31_TA01.Main.Run;
END_REGION

REGION Network 60: Station 120 - End of production
   RUNG wire#powerrail
      I_Contact( "STATUS_120".GL01_MA02.Main.Run )
      I_Contact( "STATUS_120".UH31_TA01.Main.Run )
      Contact( "STATUS_120".GL01_MA01_HomePos )
      { S7_Templates := "SrcType := Int" } EQ_Contact(in1 := "STATUS_120".PartCounter, in2 := 0)
      Coil( #TS_Station120.EndOfProd )
   END_RUNG
   // the same network as SCL:
   #TS_Station120.EndOfProd := NOT "STATUS_120".GL01_MA02.Main.Run AND NOT "STATUS_120".UH31_TA01.Main.Run AND "STATUS_120".GL01_MA01_HomePos AND ("STATUS_120".PartCounter = 0);
END_REGION

REGION Network 61: Station 120 - Request End of cycle
   RUNG wire#powerrail
      Contact( "STATUS_Zone100"."RU01-QQ02".Specific.RequestUnlock )
      Coil( #TS_Station120.ReqEndOfCycle )
   END_RUNG
   // the same network as SCL:
   #TS_Station120.ReqEndOfCycle := "STATUS_Zone100"."RU01-QQ02".Specific.RequestUnlock;
END_REGION

REGION Network 62: Station 120 - Stop
   RUNG wire#powerrail
      Contact( "STATUS_120".SF04_12 )
      wire#w1
      Coil( #TS_Station120.Stop )
   END_RUNG
   RUNG wire#powerrail
      Contact( "STATUS_Zone100"."RU01-QQ02".Specific.RequestPause )
   END_RUNG wire#w1
   // the same network as SCL:
   #TS_Station120.Stop := "STATUS_120".SF04_12 OR "STATUS_Zone100"."RU01-QQ02".Specific.RequestPause;
END_REGION

REGION Network 63: Station 120 - Number of selected devices
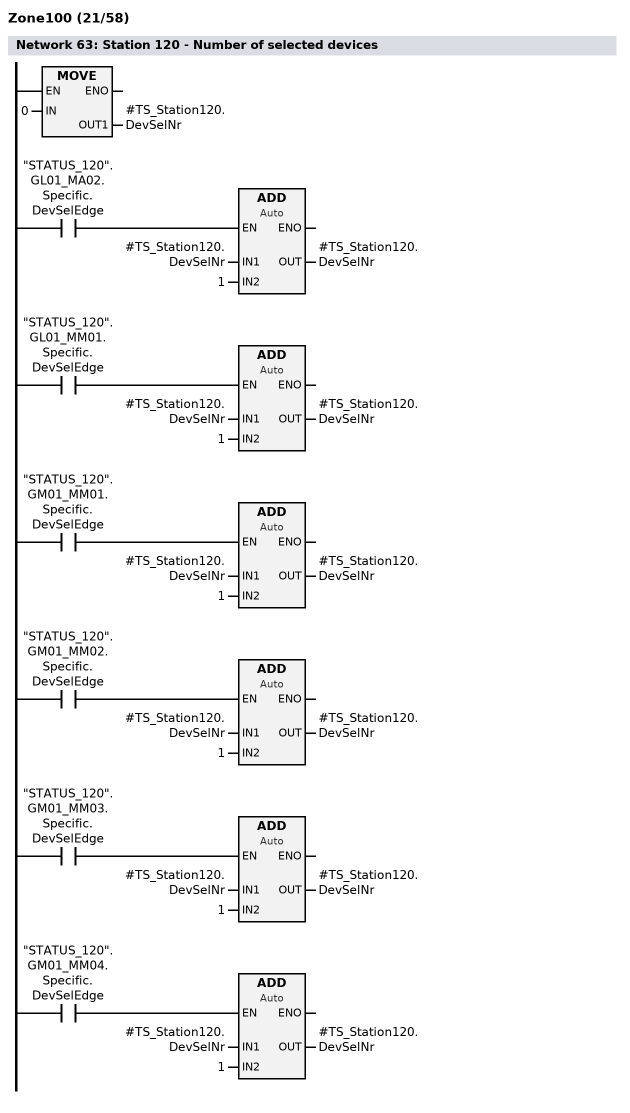
   RUNG wire#powerrail
      Move(in := 0, out1 => #TS_Station120.DevSelNr)
   END_RUNG
   RUNG wire#powerrail
      Contact( "STATUS_120".GL01_MA02.Specific.DevSelEdge )
      Add(in1 := #TS_Station120.DevSelNr, in2 := 1, out => #TS_Station120.DevSelNr)
   END_RUNG
   RUNG wire#powerrail
      Contact( "STATUS_120".GL01_MM01.Specific.DevSelEdge )
      Add(in1 := #TS_Station120.DevSelNr, in2 := 1, out => #TS_Station120.DevSelNr)
   END_RUNG
   RUNG wire#powerrail
      Contact( "STATUS_120".GM01_MM01.Specific.DevSelEdge )
      Add(in1 := #TS_Station120.DevSelNr, in2 := 1, out => #TS_Station120.DevSelNr)
   END_RUNG
   RUNG wire#powerrail
      Contact( "STATUS_120".GM01_MM02.Specific.DevSelEdge )
      Add(in1 := #TS_Station120.DevSelNr, in2 := 1, out => #TS_Station120.DevSelNr)
   END_RUNG
   RUNG wire#powerrail
      Contact( "STATUS_120".GM01_MM03.Specific.DevSelEdge )
      Add(in1 := #TS_Station120.DevSelNr, in2 := 1, out => #TS_Station120.DevSelNr)
   END_RUNG
   RUNG wire#powerrail
      Contact( "STATUS_120".GM01_MM04.Specific.DevSelEdge )
      Add(in1 := #TS_Station120.DevSelNr, in2 := 1, out => #TS_Station120.DevSelNr)
   END_RUNG
   // the same network as SCL:
   #TS_Station120.DevSelNr := 0;
   IF "STATUS_120".GL01_MA02.Specific.DevSelEdge THEN
       #TS_Station120.DevSelNr := #TS_Station120.DevSelNr + 1;
   END_IF;
   IF "STATUS_120".GL01_MM01.Specific.DevSelEdge THEN
       #TS_Station120.DevSelNr := #TS_Station120.DevSelNr + 1;
   END_IF;
   IF "STATUS_120".GM01_MM01.Specific.DevSelEdge THEN
       #TS_Station120.DevSelNr := #TS_Station120.DevSelNr + 1;
   END_IF;
   IF "STATUS_120".GM01_MM02.Specific.DevSelEdge THEN
       #TS_Station120.DevSelNr := #TS_Station120.DevSelNr + 1;
   END_IF;
   IF "STATUS_120".GM01_MM03.Specific.DevSelEdge THEN
       #TS_Station120.DevSelNr := #TS_Station120.DevSelNr + 1;
   END_IF;
   IF "STATUS_120".GM01_MM04.Specific.DevSelEdge THEN
       #TS_Station120.DevSelNr := #TS_Station120.DevSelNr + 1;
   END_IF;
END_REGION

REGION Network 64: Station 120 - Main control
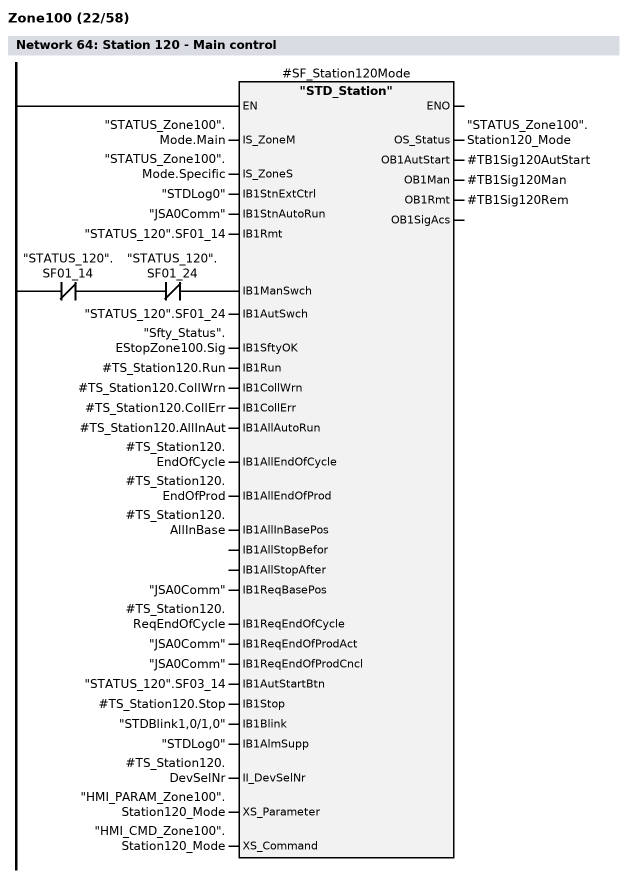
   RUNG wire#powerrail
      #SF_Station120Mode(IB1ManSwch := wire#w1, IS_ZoneM := "STATUS_Zone100".Mode.Main, IS_ZoneS := "STATUS_Zone100".Mode.Specific, IB1StnExtCtrl := "STDLog0", IB1StnAutoRun := "JSA0Comm", IB1Rmt := "STATUS_120".SF01_14, IB1AutSwch := "STATUS_120".SF01_24, IB1SftyOK := "Sfty_Status".EStopZone100.Sig, IB1Run := #TS_Station120.Run, IB1CollWrn := #TS_Station120.CollWrn, IB1CollErr := #TS_Station120.CollErr, IB1AllAutoRun := #TS_Station120.AllInAut, IB1AllEndOfCycle := #TS_Station120.EndOfCycle, IB1AllEndOfProd := #TS_Station120.EndOfProd, IB1AllInBasePos := #TS_Station120.AllInBase, IB1AllStopBefor :=, IB1AllStopAfter :=, IB1ReqBasePos := "JSA0Comm", IB1ReqEndOfCycle := #TS_Station120.ReqEndOfCycle, IB1ReqEndOfProdAct := "JSA0Comm", IB1ReqEndOfProdCncl := "JSA0Comm", IB1AutStartBtn := "STATUS_120".SF03_14, IB1Stop := #TS_Station120.Stop, IB1Blink := "STDBlink1,0/1,0", IB1AlmSupp := "STDLog0", II_DevSelNr := #TS_Station120.DevSelNr, XS_Parameter := "HMI_PARAM_Zone100".Station120_Mode, XS_Command := "HMI_CMD_Zone100".Station120_Mode, OS_Status => "STATUS_Zone100".Station120_Mode, OB1AutStart => #TB1Sig120AutStart, OB1Man => #TB1Sig120Man, OB1Rmt => #TB1Sig120Rem, OB1SigAcs =>)
   END_RUNG
   RUNG wire#powerrail
      I_Contact( "STATUS_120".SF01_14 )
      I_Contact( "STATUS_120".SF01_24 )
   END_RUNG wire#w1
   // the same network as SCL:
   #SF_Station120Mode(IS_ZoneM := "STATUS_Zone100".Mode.Main,   // "STD_Station"
                      IS_ZoneS := "STATUS_Zone100".Mode.Specific,
                      IB1StnExtCtrl := "STDLog0",
                      IB1StnAutoRun := "JSA0Comm",
                      IB1Rmt := "STATUS_120".SF01_14,
                      IB1ManSwch := NOT "STATUS_120".SF01_14 AND NOT "STATUS_120".SF01_24,
                      IB1AutSwch := "STATUS_120".SF01_24,
                      IB1SftyOK := "Sfty_Status".EStopZone100.Sig,
                      IB1Run := #TS_Station120.Run,
                      IB1CollWrn := #TS_Station120.CollWrn,
                      IB1CollErr := #TS_Station120.CollErr,
                      IB1AllAutoRun := #TS_Station120.AllInAut,
                      IB1AllEndOfCycle := #TS_Station120.EndOfCycle,
                      IB1AllEndOfProd := #TS_Station120.EndOfProd,
                      IB1AllInBasePos := #TS_Station120.AllInBase,
                      IB1ReqBasePos := "JSA0Comm",
                      IB1ReqEndOfCycle := #TS_Station120.ReqEndOfCycle,
                      IB1ReqEndOfProdAct := "JSA0Comm",
                      IB1ReqEndOfProdCncl := "JSA0Comm",
                      IB1AutStartBtn := "STATUS_120".SF03_14,
                      IB1Stop := #TS_Station120.Stop,
                      IB1Blink := "STDBlink1,0/1,0",
                      IB1AlmSupp := "STDLog0",
                      II_DevSelNr := #TS_Station120.DevSelNr,
                      XS_Parameter := "HMI_PARAM_Zone100".Station120_Mode,
                      XS_Command := "HMI_CMD_Zone100".Station120_Mode,
                      OS_Status => "STATUS_Zone100".Station120_Mode,
                      OB1AutStart => #TB1Sig120AutStart,
                      OB1Man => #TB1Sig120Man,
                      OB1Rmt => #TB1Sig120Rem);
END_REGION

